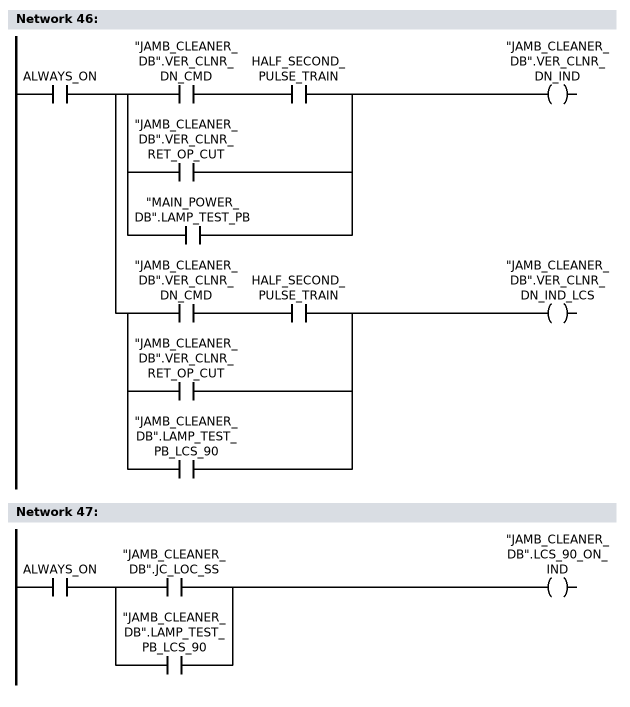
NETWORK
TITLE =
      A     "ALWAYS_ON";
      =     L 0.0;
      A     L 0.0;
      A(;
      A     "JAMB_CLEANER_DB".VER_CLNR_DN_CMD;
      A     "HALF_SECOND_PULSE_TRAIN";
      O     "JAMB_CLEANER_DB".VER_CLNR_RET_OP_CUT;
      O     "MAIN_POWER_DB".LAMP_TEST_PB;
      );
      =     "JAMB_CLEANER_DB".VER_CLNR_DN_IND;
      A     L 0.0;
      A(;
      A     "JAMB_CLEANER_DB".VER_CLNR_DN_CMD;
      A     "HALF_SECOND_PULSE_TRAIN";
      O     "JAMB_CLEANER_DB".VER_CLNR_RET_OP_CUT;
      O     "JAMB_CLEANER_DB".LAMP_TEST_PB_LCS_90;
      );
      =     "JAMB_CLEANER_DB".VER_CLNR_DN_IND_LCS;
NETWORK
TITLE =
      A     "ALWAYS_ON";
      A(;
      O     "JAMB_CLEANER_DB".JC_LOC_SS;
      O     "JAMB_CLEANER_DB".LAMP_TEST_PB_LCS_90;
      );
      =     "JAMB_CLEANER_DB".LCS_90_ON_IND;
END_FUNCTION

FUNCTION "COUNTER_THRUST_WEDGE" : VOID	// FC 17
AUTHOR : Kamillas
VERSION : 0.1
BEGIN
// (block stored without names or comments; labels and parameter names are numbered)
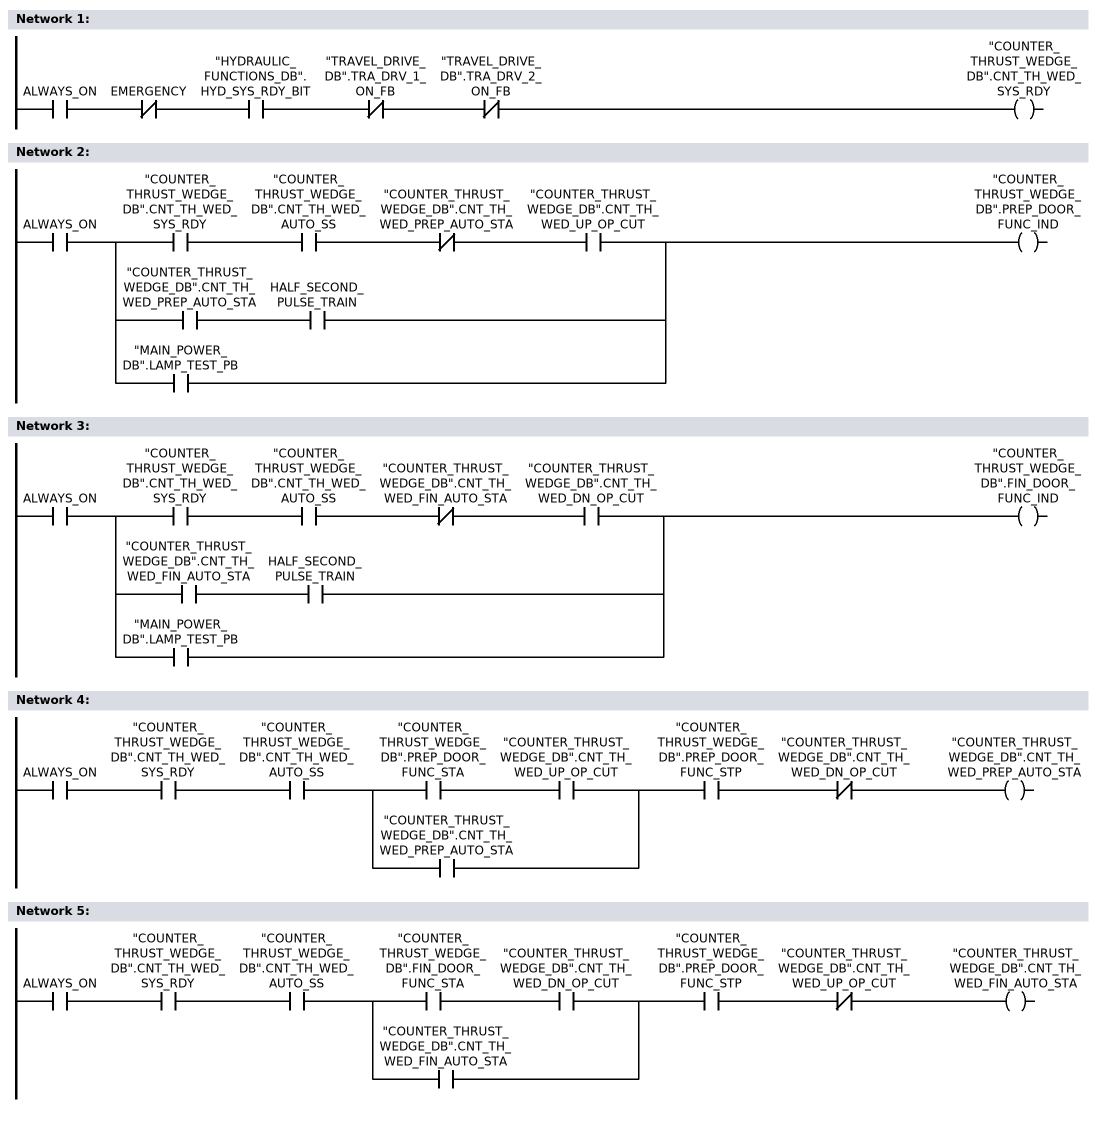
NETWORK
TITLE =
      A     "ALWAYS_ON";
      AN    "EMERGENCY";
      A     "HYDRAULIC_FUNCTIONS_DB".HYD_SYS_RDY_BIT;
      AN    "TRAVEL_DRIVE_DB".TRA_DRV_1_ON_FB;
      AN    "TRAVEL_DRIVE_DB".TRA_DRV_2_ON_FB;
      =     "COUNTER_THRUST_WEDGE_DB".CNT_TH_WED_SYS_RDY;
NETWORK
TITLE =
      A     "ALWAYS_ON";
      A(;
      A     "COUNTER_THRUST_WEDGE_DB".CNT_TH_WED_SYS_RDY;
      A     "COUNTER_THRUST_WEDGE_DB".CNT_TH_WED_AUTO_SS;
      AN    "COUNTER_THRUST_WEDGE_DB".CNT_TH_WED_PREP_AUTO_STA;
      A     "COUNTER_THRUST_WEDGE_DB".CNT_TH_WED_UP_OP_CUT;
      O;
      A     "COUNTER_THRUST_WEDGE_DB".CNT_TH_WED_PREP_AUTO_STA;
      A     "HALF_SECOND_PULSE_TRAIN";
      O     "MAIN_POWER_DB".LAMP_TEST_PB;
      );
      =     "COUNTER_THRUST_WEDGE_DB".PREP_DOOR_FUNC_IND;
NETWORK
TITLE =
      A     "ALWAYS_ON";
      A(;
      A     "COUNTER_THRUST_WEDGE_DB".CNT_TH_WED_SYS_RDY;
      A     "COUNTER_THRUST_WEDGE_DB".CNT_TH_WED_AUTO_SS;
      AN    "COUNTER_THRUST_WEDGE_DB".CNT_TH_WED_FIN_AUTO_STA;
      A     "COUNTER_THRUST_WEDGE_DB".CNT_TH_WED_DN_OP_CUT;
      O;
      A     "COUNTER_THRUST_WEDGE_DB".CNT_TH_WED_FIN_AUTO_STA;
      A     "HALF_SECOND_PULSE_TRAIN";
      O     "MAIN_POWER_DB".LAMP_TEST_PB;
      );
      =     "COUNTER_THRUST_WEDGE_DB".FIN_DOOR_FUNC_IND;
NETWORK
TITLE =
      A     "ALWAYS_ON";
      A     "COUNTER_THRUST_WEDGE_DB".CNT_TH_WED_SYS_RDY;
      A     "COUNTER_THRUST_WEDGE_DB".CNT_TH_WED_AUTO_SS;
      A(;
      A     "COUNTER_THRUST_WEDGE_DB".PREP_DOOR_FUNC_STA;
      A     "COUNTER_THRUST_WEDGE_DB".CNT_TH_WED_UP_OP_CUT;
      O     "COUNTER_THRUST_WEDGE_DB".CNT_TH_WED_PREP_AUTO_STA;
      );
      A     "COUNTER_THRUST_WEDGE_DB".PREP_DOOR_FUNC_STP;
      AN    "COUNTER_THRUST_WEDGE_DB".CNT_TH_WED_DN_OP_CUT;
      =     "COUNTER_THRUST_WEDGE_DB".CNT_TH_WED_PREP_AUTO_STA;
NETWORK
TITLE =
      A     "ALWAYS_ON";
      A     "COUNTER_THRUST_WEDGE_DB".CNT_TH_WED_SYS_RDY;
      A     "COUNTER_THRUST_WEDGE_DB".CNT_TH_WED_AUTO_SS;
      A(;
      A     "COUNTER_THRUST_WEDGE_DB".FIN_DOOR_FUNC_STA;
      A     "COUNTER_THRUST_WEDGE_DB".CNT_TH_WED_DN_OP_CUT;
      O     "COUNTER_THRUST_WEDGE_DB".CNT_TH_WED_FIN_AUTO_STA;
      );
      A     "COUNTER_THRUST_WEDGE_DB".PREP_DOOR_FUNC_STP;
      AN    "COUNTER_THRUST_WEDGE_DB".CNT_TH_WED_UP_OP_CUT;
      =     "COUNTER_THRUST_WEDGE_DB".CNT_TH_WED_FIN_AUTO_STA;
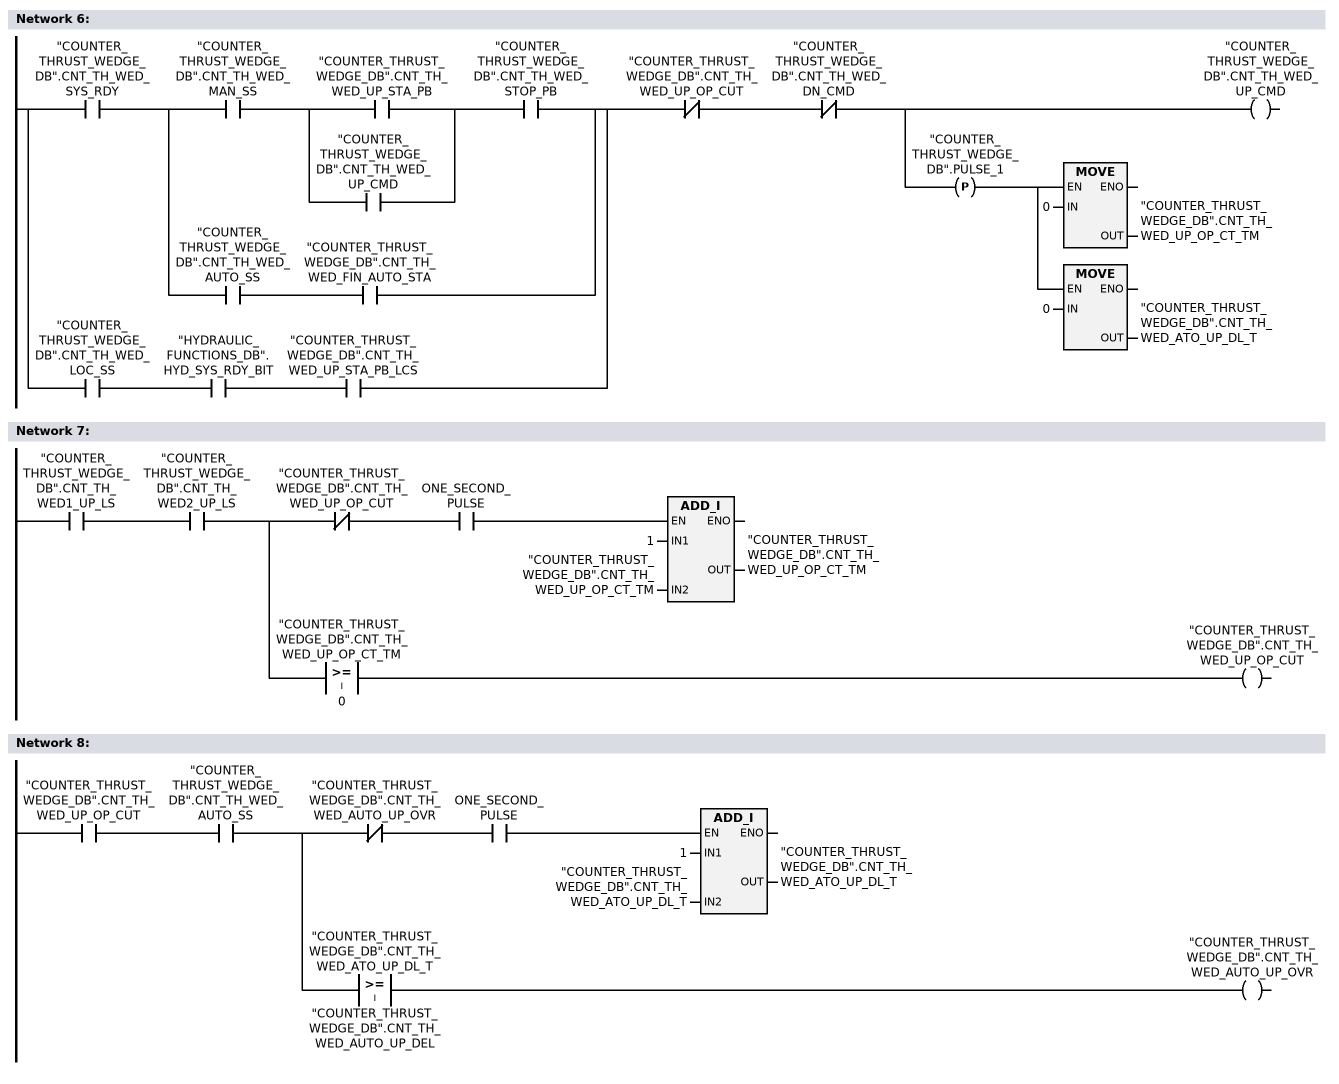
NETWORK
TITLE =
      A(;
      A     "COUNTER_THRUST_WEDGE_DB".CNT_TH_WED_SYS_RDY;
      A(;
      A     "COUNTER_THRUST_WEDGE_DB".CNT_TH_WED_MAN_SS;
      A(;
      O     "COUNTER_THRUST_WEDGE_DB".CNT_TH_WED_UP_STA_PB;
      O     "COUNTER_THRUST_WEDGE_DB".CNT_TH_WED_UP_CMD;
      );
      A     "COUNTER_THRUST_WEDGE_DB".CNT_TH_WED_STOP_PB;
      O;
      A     "COUNTER_THRUST_WEDGE_DB".CNT_TH_WED_AUTO_SS;
      A     "COUNTER_THRUST_WEDGE_DB".CNT_TH_WED_FIN_AUTO_STA;
      );
      O;
      A     "COUNTER_THRUST_WEDGE_DB".CNT_TH_WED_LOC_SS;
      A     "HYDRAULIC_FUNCTIONS_DB".HYD_SYS_RDY_BIT;
      A     "COUNTER_THRUST_WEDGE_DB".CNT_TH_WED_UP_STA_PB_LCS;
      );
      AN    "COUNTER_THRUST_WEDGE_DB".CNT_TH_WED_UP_OP_CUT;
      AN    "COUNTER_THRUST_WEDGE_DB".CNT_TH_WED_DN_CMD;
      =     L 0.0;
      A     L 0.0;
      BLD   102;
      =     "COUNTER_THRUST_WEDGE_DB".CNT_TH_WED_UP_CMD;
      A     L 0.0;
      FP    "COUNTER_THRUST_WEDGE_DB".PULSE_1;
      =     L 0.1;
      A     L 0.1;
      JNB   M001;
      L     0;
      T     "COUNTER_THRUST_WEDGE_DB".CNT_TH_WED_UP_OP_CT_TM;
M001: NOP   0;
      A     L 0.1;
      JNB   M002;
      L     0;
      T     "COUNTER_THRUST_WEDGE_DB".CNT_TH_WED_ATO_UP_DL_T;
M002: NOP   0;
NETWORK
TITLE =
      A     "COUNTER_THRUST_WEDGE_DB".CNT_TH_WED1_UP_LS;
      A     "COUNTER_THRUST_WEDGE_DB".CNT_TH_WED2_UP_LS;
      =     L 0.0;
      A     L 0.0;
      AN    "COUNTER_THRUST_WEDGE_DB".CNT_TH_WED_UP_OP_CUT;
      A     "ONE_SECOND_PULSE";
      JNB   M003;
      L     1;
      L     "COUNTER_THRUST_WEDGE_DB".CNT_TH_WED_UP_OP_CT_TM;
      +I;
      T     "COUNTER_THRUST_WEDGE_DB".CNT_TH_WED_UP_OP_CT_TM;
M003: NOP   0;
      A     L 0.0;
      A(;
      L     "COUNTER_THRUST_WEDGE_DB".CNT_TH_WED_UP_OP_CT_TM;
      L     0;
      >=I;
      );
      =     "COUNTER_THRUST_WEDGE_DB".CNT_TH_WED_UP_OP_CUT;
NETWORK
TITLE =
      A     "COUNTER_THRUST_WEDGE_DB".CNT_TH_WED_UP_OP_CUT;
      A     "COUNTER_THRUST_WEDGE_DB".CNT_TH_WED_AUTO_SS;
      =     L 0.0;
      A     L 0.0;
      AN    "COUNTER_THRUST_WEDGE_DB".CNT_TH_WED_AUTO_UP_OVR;
      A     "ONE_SECOND_PULSE";
      JNB   M004;
      L     1;
      L     "COUNTER_THRUST_WEDGE_DB".CNT_TH_WED_ATO_UP_DL_T;
      +I;
      T     "COUNTER_THRUST_WEDGE_DB".CNT_TH_WED_ATO_UP_DL_T;
M004: NOP   0;
      A     L 0.0;
      A(;
      L     "COUNTER_THRUST_WEDGE_DB".CNT_TH_WED_ATO_UP_DL_T;
      L     "COUNTER_THRUST_WEDGE_DB".CNT_TH_WED_AUTO_UP_DEL;
      >=I;
      );
      =     "COUNTER_THRUST_WEDGE_DB".CNT_TH_WED_AUTO_UP_OVR;
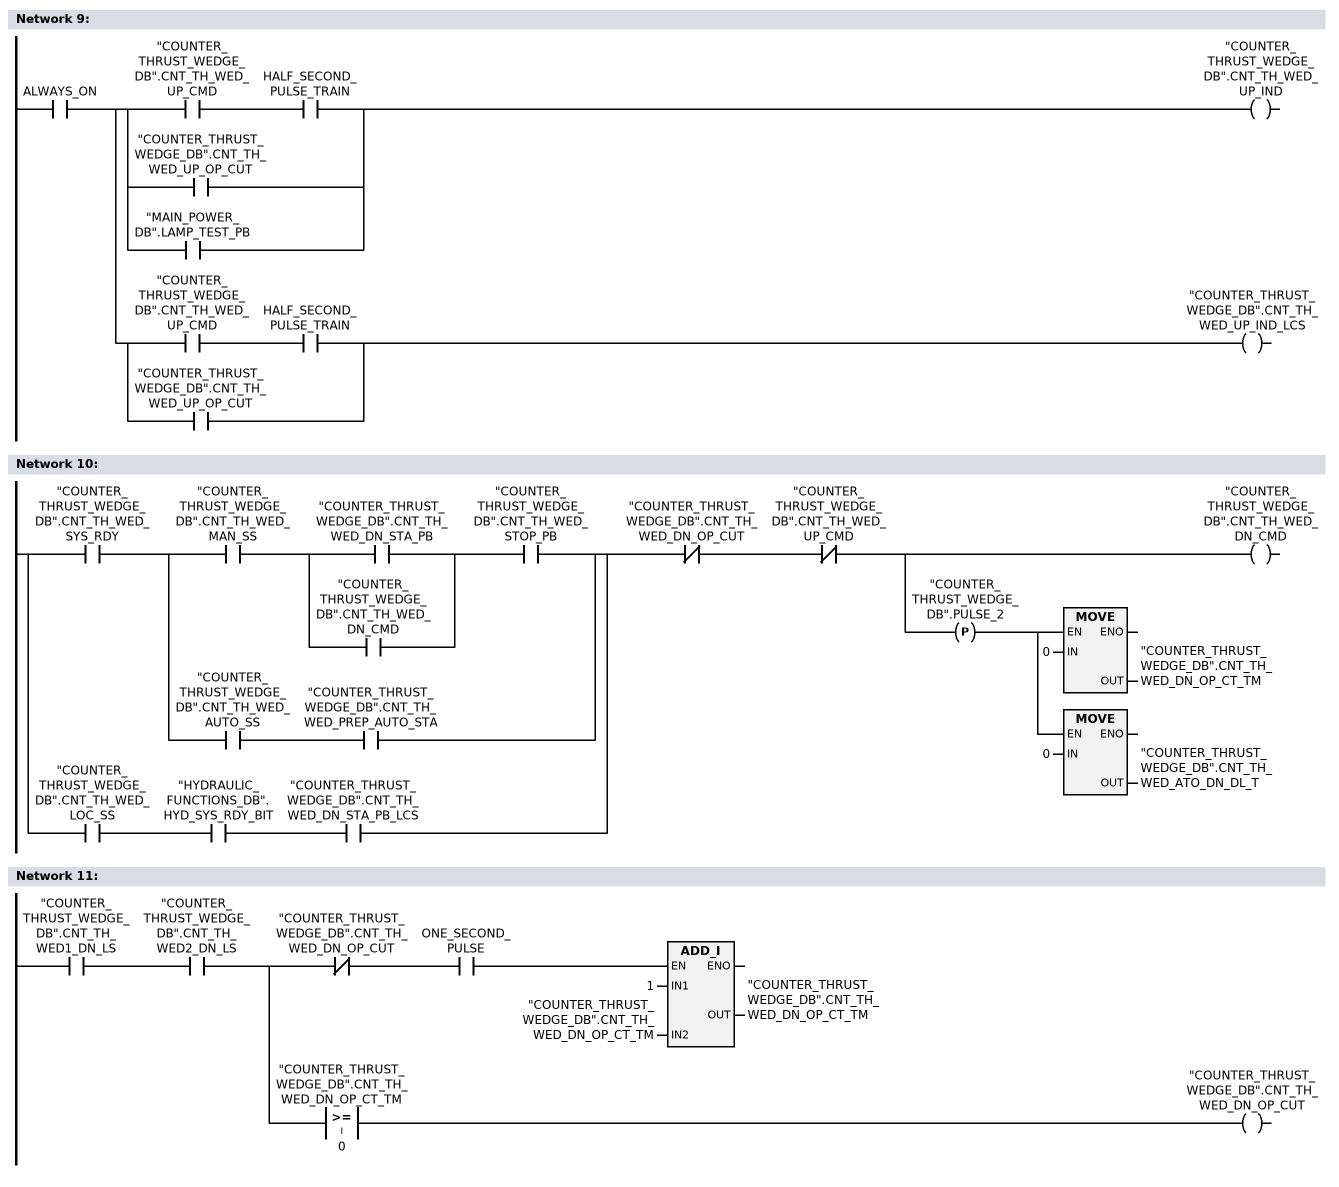
NETWORK
TITLE =
      A     "ALWAYS_ON";
      =     L 0.0;
      A     L 0.0;
      A(;
      A     "COUNTER_THRUST_WEDGE_DB".CNT_TH_WED_UP_CMD;
      A     "HALF_SECOND_PULSE_TRAIN";
      O     "COUNTER_THRUST_WEDGE_DB".CNT_TH_WED_UP_OP_CUT;
      O     "MAIN_POWER_DB".LAMP_TEST_PB;
      );
      =     "COUNTER_THRUST_WEDGE_DB".CNT_TH_WED_UP_IND;
      A     L 0.0;
      A(;
      A     "COUNTER_THRUST_WEDGE_DB".CNT_TH_WED_UP_CMD;
      A     "HALF_SECOND_PULSE_TRAIN";
      O     "COUNTER_THRUST_WEDGE_DB".CNT_TH_WED_UP_OP_CUT;
      );
      =     "COUNTER_THRUST_WEDGE_DB".CNT_TH_WED_UP_IND_LCS;
NETWORK
TITLE =
      A(;
      A     "COUNTER_THRUST_WEDGE_DB".CNT_TH_WED_SYS_RDY;
      A(;
      A     "COUNTER_THRUST_WEDGE_DB".CNT_TH_WED_MAN_SS;
      A(;
      O     "COUNTER_THRUST_WEDGE_DB".CNT_TH_WED_DN_STA_PB;
      O     "COUNTER_THRUST_WEDGE_DB".CNT_TH_WED_DN_CMD;
      );
      A     "COUNTER_THRUST_WEDGE_DB".CNT_TH_WED_STOP_PB;
      O;
      A     "COUNTER_THRUST_WEDGE_DB".CNT_TH_WED_AUTO_SS;
      A     "COUNTER_THRUST_WEDGE_DB".CNT_TH_WED_PREP_AUTO_STA;
      );
      O;
      A     "COUNTER_THRUST_WEDGE_DB".CNT_TH_WED_LOC_SS;
      A     "HYDRAULIC_FUNCTIONS_DB".HYD_SYS_RDY_BIT;
      A     "COUNTER_THRUST_WEDGE_DB".CNT_TH_WED_DN_STA_PB_LCS;
      );
      AN    "COUNTER_THRUST_WEDGE_DB".CNT_TH_WED_DN_OP_CUT;
      AN    "COUNTER_THRUST_WEDGE_DB".CNT_TH_WED_UP_CMD;
      =     L 0.0;
      A     L 0.0;
      BLD   102;
      =     "COUNTER_THRUST_WEDGE_DB".CNT_TH_WED_DN_CMD;
      A     L 0.0;
      FP    "COUNTER_THRUST_WEDGE_DB".PULSE_2;
      =     L 0.1;
      A     L 0.1;
      JNB   M005;
      L     0;
      T     "COUNTER_THRUST_WEDGE_DB".CNT_TH_WED_DN_OP_CT_TM;
M005: NOP   0;
      A     L 0.1;
      JNB   M006;
      L     0;
      T     "COUNTER_THRUST_WEDGE_DB".CNT_TH_WED_ATO_DN_DL_T;
M006: NOP   0;
NETWORK
TITLE =
      A     "COUNTER_THRUST_WEDGE_DB".CNT_TH_WED1_DN_LS;
      A     "COUNTER_THRUST_WEDGE_DB".CNT_TH_WED2_DN_LS;
      =     L 0.0;
      A     L 0.0;
      AN    "COUNTER_THRUST_WEDGE_DB".CNT_TH_WED_DN_OP_CUT;
      A     "ONE_SECOND_PULSE";
      JNB   M007;
      L     1;
      L     "COUNTER_THRUST_WEDGE_DB".CNT_TH_WED_DN_OP_CT_TM;
      +I;
      T     "COUNTER_THRUST_WEDGE_DB".CNT_TH_WED_DN_OP_CT_TM;
M007: NOP   0;
      A     L 0.0;
      A(;
      L     "COUNTER_THRUST_WEDGE_DB".CNT_TH_WED_DN_OP_CT_TM;
      L     0;
      >=I;
      );
      =     "COUNTER_THRUST_WEDGE_DB".CNT_TH_WED_DN_OP_CUT;
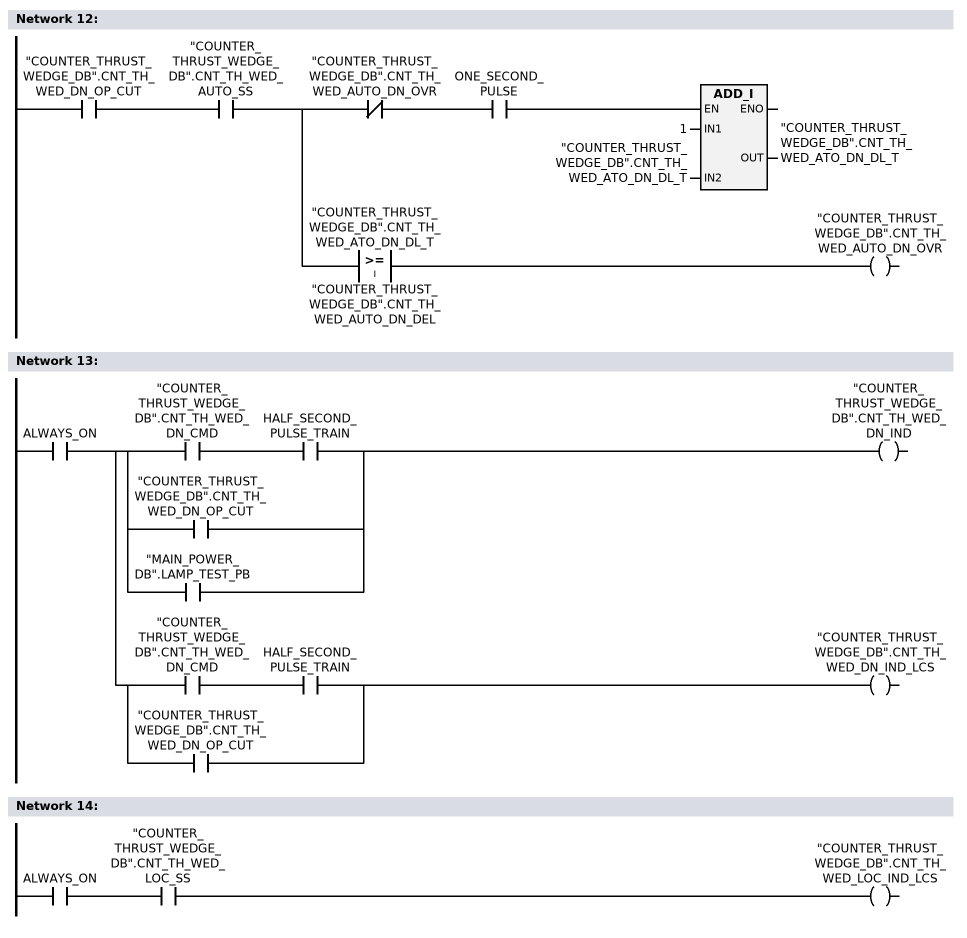
NETWORK
TITLE =
      A     "COUNTER_THRUST_WEDGE_DB".CNT_TH_WED_DN_OP_CUT;
      A     "COUNTER_THRUST_WEDGE_DB".CNT_TH_WED_AUTO_SS;
      =     L 0.0;
      A     L 0.0;
      AN    "COUNTER_THRUST_WEDGE_DB".CNT_TH_WED_AUTO_DN_OVR;
      A     "ONE_SECOND_PULSE";
      JNB   M008;
      L     1;
      L     "COUNTER_THRUST_WEDGE_DB".CNT_TH_WED_ATO_DN_DL_T;
      +I;
      T     "COUNTER_THRUST_WEDGE_DB".CNT_TH_WED_ATO_DN_DL_T;
M008: NOP   0;
      A     L 0.0;
      A(;
      L     "COUNTER_THRUST_WEDGE_DB".CNT_TH_WED_ATO_DN_DL_T;
      L     "COUNTER_THRUST_WEDGE_DB".CNT_TH_WED_AUTO_DN_DEL;
      >=I;
      );
      =     "COUNTER_THRUST_WEDGE_DB".CNT_TH_WED_AUTO_DN_OVR;
NETWORK
TITLE =
      A     "ALWAYS_ON";
      =     L 0.0;
      A     L 0.0;
      A(;
      A     "COUNTER_THRUST_WEDGE_DB".CNT_TH_WED_DN_CMD;
      A     "HALF_SECOND_PULSE_TRAIN";
      O     "COUNTER_THRUST_WEDGE_DB".CNT_TH_WED_DN_OP_CUT;
      O     "MAIN_POWER_DB".LAMP_TEST_PB;
      );
      =     "COUNTER_THRUST_WEDGE_DB".CNT_TH_WED_DN_IND;
      A     L 0.0;
      A(;
      A     "COUNTER_THRUST_WEDGE_DB".CNT_TH_WED_DN_CMD;
      A     "HALF_SECOND_PULSE_TRAIN";
      O     "COUNTER_THRUST_WEDGE_DB".CNT_TH_WED_DN_OP_CUT;
      );
      =     "COUNTER_THRUST_WEDGE_DB".CNT_TH_WED_DN_IND_LCS;
NETWORK
TITLE =
      A     "ALWAYS_ON";
      A     "COUNTER_THRUST_WEDGE_DB".CNT_TH_WED_LOC_SS;
      =     "COUNTER_THRUST_WEDGE_DB".CNT_TH_WED_LOC_IND_LCS;
END_FUNCTION

FUNCTION "COAL_SPILLAGE_SYSTEM" : VOID	// FC 18
AUTHOR : Kamillas
VERSION : 0.1
BEGIN
// (block stored without names or comments; labels and parameter names are numbered)
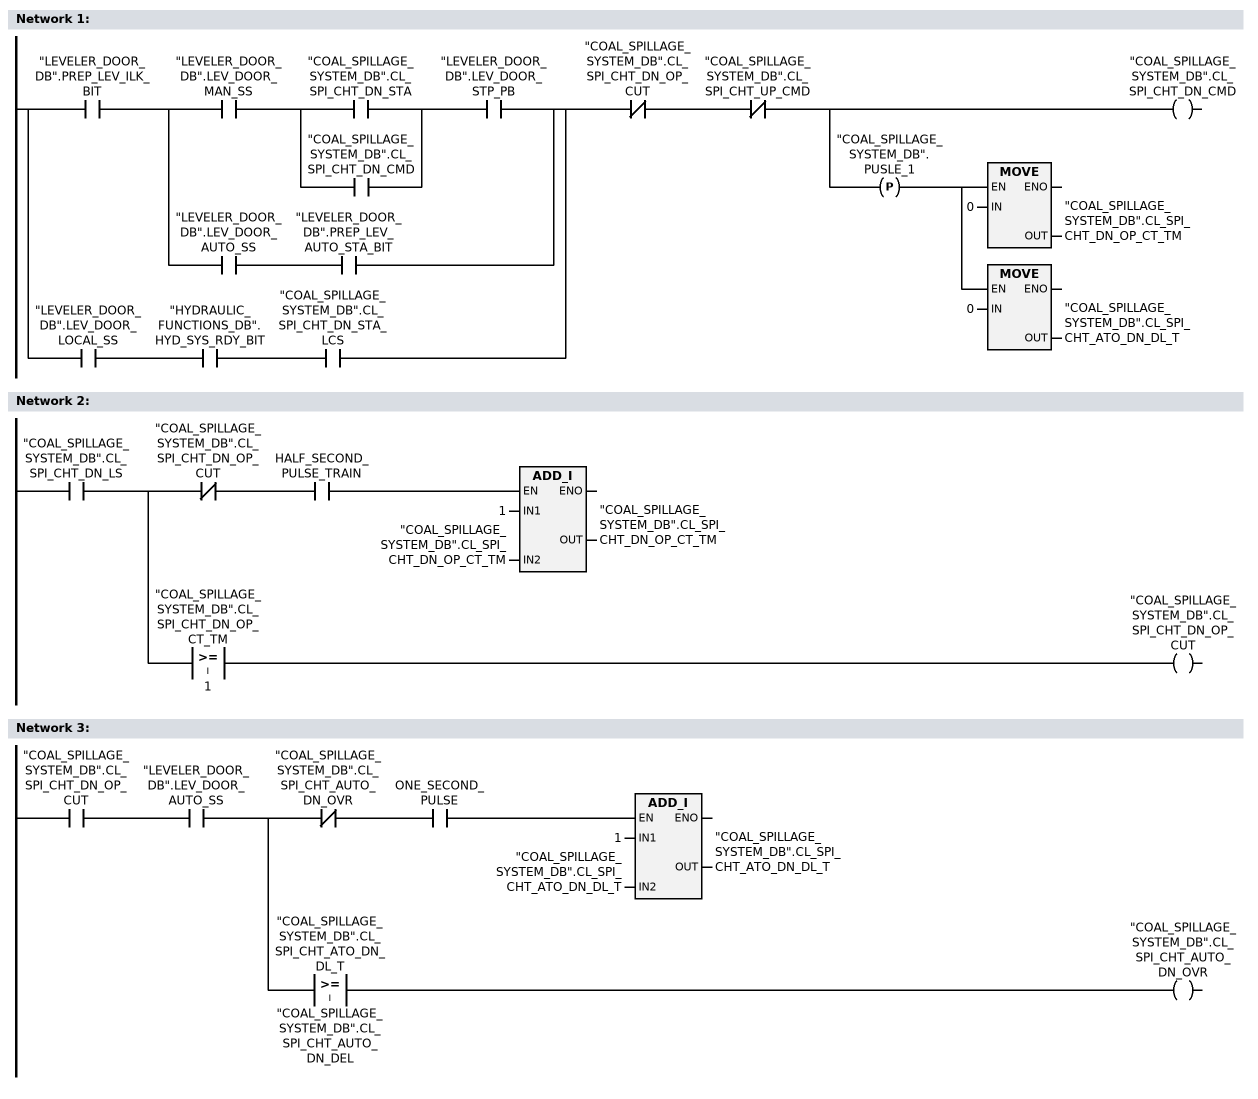
NETWORK
TITLE =
      A(;
      A     "LEVELER_DOOR_DB".PREP_LEV_ILK_BIT;
      A(;
      A     "LEVELER_DOOR_DB".LEV_DOOR_MAN_SS;
      A(;
      O     "COAL_SPILLAGE_SYSTEM_DB".CL_SPI_CHT_DN_STA;
      O     "COAL_SPILLAGE_SYSTEM_DB".CL_SPI_CHT_DN_CMD;
      );
      A     "LEVELER_DOOR_DB".LEV_DOOR_STP_PB;
      O;
      A     "LEVELER_DOOR_DB".LEV_DOOR_AUTO_SS;
      A     "LEVELER_DOOR_DB".PREP_LEV_AUTO_STA_BIT;
      );
      O;
      A     "LEVELER_DOOR_DB".LEV_DOOR_LOCAL_SS;
      A     "HYDRAULIC_FUNCTIONS_DB".HYD_SYS_RDY_BIT;
      A     "COAL_SPILLAGE_SYSTEM_DB".CL_SPI_CHT_DN_STA_LCS;
      );
      AN    "COAL_SPILLAGE_SYSTEM_DB".CL_SPI_CHT_DN_OP_CUT;
      AN    "COAL_SPILLAGE_SYSTEM_DB".CL_SPI_CHT_UP_CMD;
      =     L 0.0;
      A     L 0.0;
      BLD   102;
      =     "COAL_SPILLAGE_SYSTEM_DB".CL_SPI_CHT_DN_CMD;
      A     L 0.0;
      FP    "COAL_SPILLAGE_SYSTEM_DB".PUSLE_1;
      =     L 0.1;
      A     L 0.1;
      JNB   M001;
      L     0;
      T     "COAL_SPILLAGE_SYSTEM_DB".CL_SPI_CHT_DN_OP_CT_TM;
M001: NOP   0;
      A     L 0.1;
      JNB   M002;
      L     0;
      T     "COAL_SPILLAGE_SYSTEM_DB".CL_SPI_CHT_ATO_DN_DL_T;
M002: NOP   0;
NETWORK
TITLE =
      A     "COAL_SPILLAGE_SYSTEM_DB".CL_SPI_CHT_DN_LS;
      =     L 0.0;
      A     L 0.0;
      AN    "COAL_SPILLAGE_SYSTEM_DB".CL_SPI_CHT_DN_OP_CUT;
      A     "HALF_SECOND_PULSE_TRAIN";
      JNB   M003;
      L     1;
      L     "COAL_SPILLAGE_SYSTEM_DB".CL_SPI_CHT_DN_OP_CT_TM;
      +I;
      T     "COAL_SPILLAGE_SYSTEM_DB".CL_SPI_CHT_DN_OP_CT_TM;
M003: NOP   0;
      A     L 0.0;
      A(;
      L     "COAL_SPILLAGE_SYSTEM_DB".CL_SPI_CHT_DN_OP_CT_TM;
      L     1;
      >=I;
      );
      =     "COAL_SPILLAGE_SYSTEM_DB".CL_SPI_CHT_DN_OP_CUT;
NETWORK
TITLE =
      A     "COAL_SPILLAGE_SYSTEM_DB".CL_SPI_CHT_DN_OP_CUT;
      A     "LEVELER_DOOR_DB".LEV_DOOR_AUTO_SS;
      =     L 0.0;
      A     L 0.0;
      AN    "COAL_SPILLAGE_SYSTEM_DB".CL_SPI_CHT_AUTO_DN_OVR;
      A     "ONE_SECOND_PULSE";
      JNB   M004;
      L     1;
      L     "COAL_SPILLAGE_SYSTEM_DB".CL_SPI_CHT_ATO_DN_DL_T;
      +I;
      T     "COAL_SPILLAGE_SYSTEM_DB".CL_SPI_CHT_ATO_DN_DL_T;
M004: NOP   0;
      A     L 0.0;
      A(;
      L     "COAL_SPILLAGE_SYSTEM_DB".CL_SPI_CHT_ATO_DN_DL_T;
      L     "COAL_SPILLAGE_SYSTEM_DB".CL_SPI_CHT_AUTO_DN_DEL;
      >=I;
      );
      =     "COAL_SPILLAGE_SYSTEM_DB".CL_SPI_CHT_AUTO_DN_OVR;
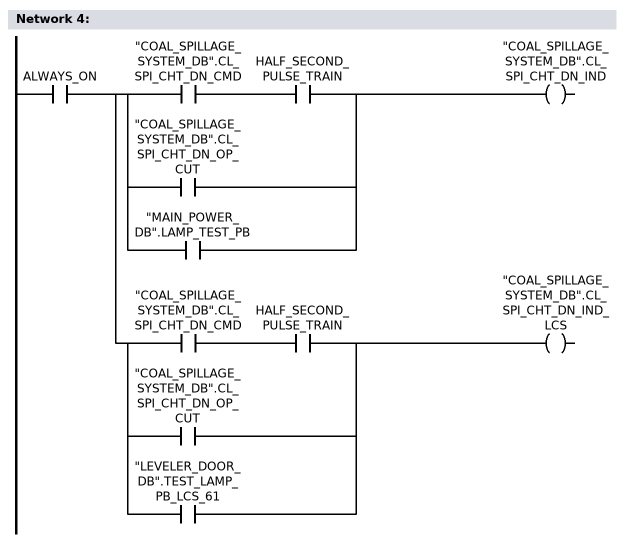
NETWORK
TITLE =
      A     "ALWAYS_ON";
      =     L 0.0;
      A     L 0.0;
      A(;
      A     "COAL_SPILLAGE_SYSTEM_DB".CL_SPI_CHT_DN_CMD;
      A     "HALF_SECOND_PULSE_TRAIN";
      O     "COAL_SPILLAGE_SYSTEM_DB".CL_SPI_CHT_DN_OP_CUT;
      O     "MAIN_POWER_DB".LAMP_TEST_PB;
      );
      =     "COAL_SPILLAGE_SYSTEM_DB".CL_SPI_CHT_DN_IND;
      A     L 0.0;
      A(;
      A     "COAL_SPILLAGE_SYSTEM_DB".CL_SPI_CHT_DN_CMD;
      A     "HALF_SECOND_PULSE_TRAIN";
      O     "COAL_SPILLAGE_SYSTEM_DB".CL_SPI_CHT_DN_OP_CUT;
      O     "LEVELER_DOOR_DB".TEST_LAMP_PB_LCS_61;
      );
      =     "COAL_SPILLAGE_SYSTEM_DB".CL_SPI_CHT_DN_IND_LCS;
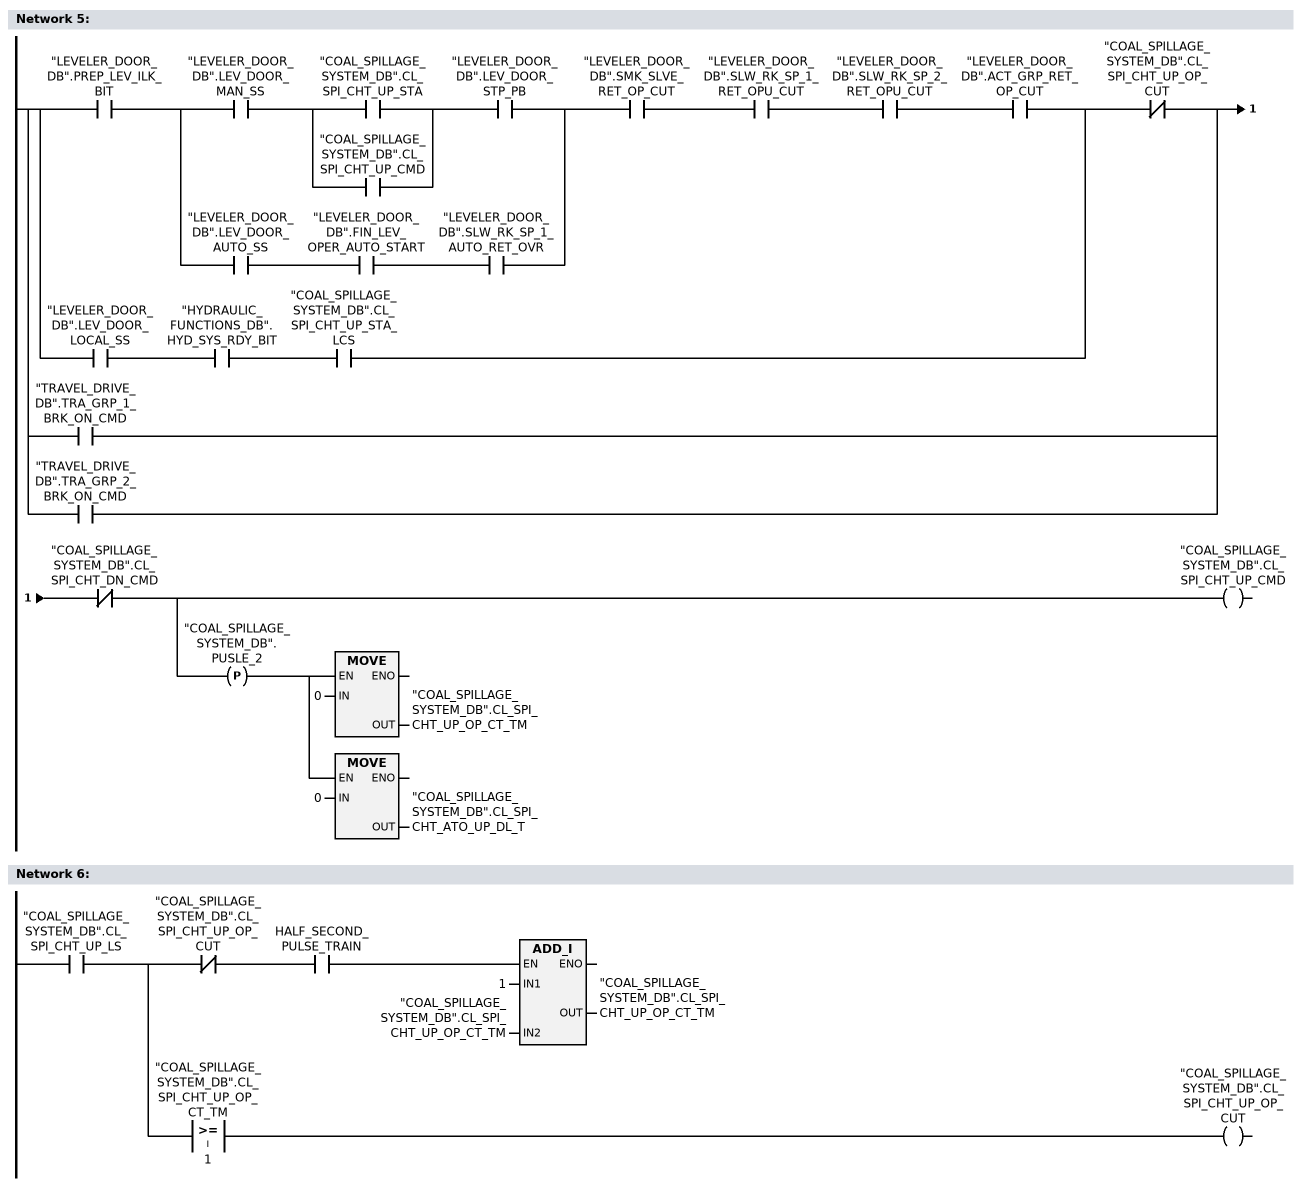
NETWORK
TITLE =
      A(;
      A(;
      A     "LEVELER_DOOR_DB".PREP_LEV_ILK_BIT;
      A(;
      A     "LEVELER_DOOR_DB".LEV_DOOR_MAN_SS;
      A(;
      O     "COAL_SPILLAGE_SYSTEM_DB".CL_SPI_CHT_UP_STA;
      O     "COAL_SPILLAGE_SYSTEM_DB".CL_SPI_CHT_UP_CMD;
      );
      A     "LEVELER_DOOR_DB".LEV_DOOR_STP_PB;
      O;
      A     "LEVELER_DOOR_DB".LEV_DOOR_AUTO_SS;
      A     "LEVELER_DOOR_DB".FIN_LEV_OPER_AUTO_START;
      A     "LEVELER_DOOR_DB".SLW_RK_SP_1_AUTO_RET_OVR;
      );
      A     "LEVELER_DOOR_DB".SMK_SLVE_RET_OP_CUT;
      A     "LEVELER_DOOR_DB".SLW_RK_SP_1_RET_OPU_CUT;
      A     "LEVELER_DOOR_DB".SLW_RK_SP_2_RET_OPU_CUT;
      A     "LEVELER_DOOR_DB".ACT_GRP_RET_OP_CUT;
      O;
      A     "LEVELER_DOOR_DB".LEV_DOOR_LOCAL_SS;
      A     "HYDRAULIC_FUNCTIONS_DB".HYD_SYS_RDY_BIT;
      A     "COAL_SPILLAGE_SYSTEM_DB".CL_SPI_CHT_UP_STA_LCS;
      );
      AN    "COAL_SPILLAGE_SYSTEM_DB".CL_SPI_CHT_UP_OP_CUT;
      O     "TRAVEL_DRIVE_DB".TRA_GRP_1_BRK_ON_CMD;
      O     "TRAVEL_DRIVE_DB".TRA_GRP_2_BRK_ON_CMD;
      );
      AN    "COAL_SPILLAGE_SYSTEM_DB".CL_SPI_CHT_DN_CMD;
      =     L 0.0;
      A     L 0.0;
      BLD   102;
      =     "COAL_SPILLAGE_SYSTEM_DB".CL_SPI_CHT_UP_CMD;
      A     L 0.0;
      FP    "COAL_SPILLAGE_SYSTEM_DB".PUSLE_2;
      =     L 0.1;
      A     L 0.1;
      JNB   M005;
      L     0;
      T     "COAL_SPILLAGE_SYSTEM_DB".CL_SPI_CHT_UP_OP_CT_TM;
M005: NOP   0;
      A     L 0.1;
      JNB   M006;
      L     0;
      T     "COAL_SPILLAGE_SYSTEM_DB".CL_SPI_CHT_ATO_UP_DL_T;
M006: NOP   0;
NETWORK
TITLE =
      A     "COAL_SPILLAGE_SYSTEM_DB".CL_SPI_CHT_UP_LS;
      =     L 0.0;
      A     L 0.0;
      AN    "COAL_SPILLAGE_SYSTEM_DB".CL_SPI_CHT_UP_OP_CUT;
      A     "HALF_SECOND_PULSE_TRAIN";
      JNB   M007;
      L     1;
      L     "COAL_SPILLAGE_SYSTEM_DB".CL_SPI_CHT_UP_OP_CT_TM;
      +I;
      T     "COAL_SPILLAGE_SYSTEM_DB".CL_SPI_CHT_UP_OP_CT_TM;
M007: NOP   0;
      A     L 0.0;
      A(;
      L     "COAL_SPILLAGE_SYSTEM_DB".CL_SPI_CHT_UP_OP_CT_TM;
      L     1;
      >=I;
      );
      =     "COAL_SPILLAGE_SYSTEM_DB".CL_SPI_CHT_UP_OP_CUT;
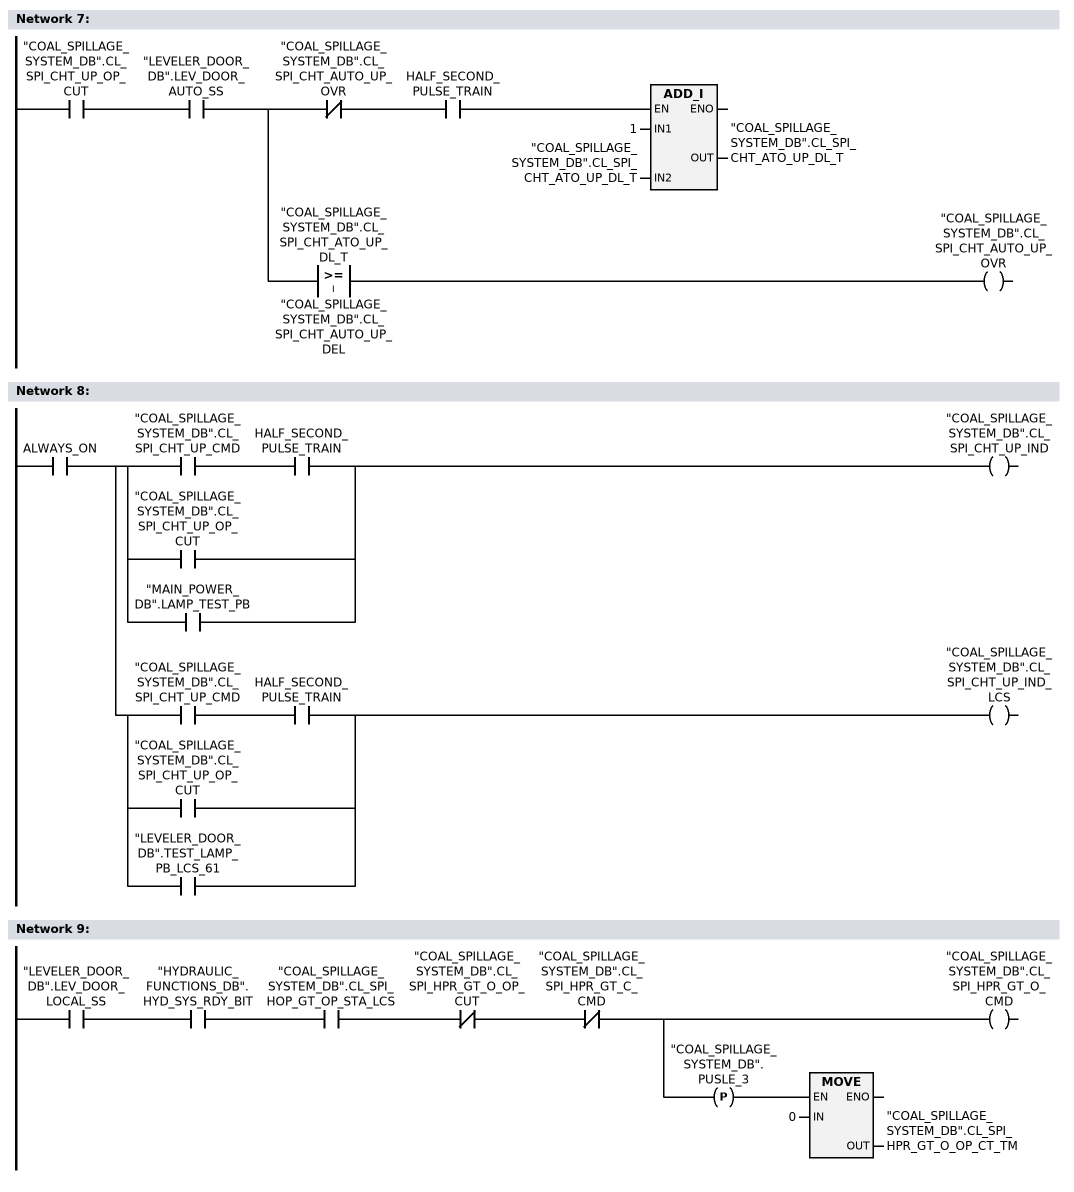
NETWORK
TITLE =
      A     "COAL_SPILLAGE_SYSTEM_DB".CL_SPI_CHT_UP_OP_CUT;
      A     "LEVELER_DOOR_DB".LEV_DOOR_AUTO_SS;
      =     L 0.0;
      A     L 0.0;
      AN    "COAL_SPILLAGE_SYSTEM_DB".CL_SPI_CHT_AUTO_UP_OVR;
      A     "HALF_SECOND_PULSE_TRAIN";
      JNB   M008;
      L     1;
      L     "COAL_SPILLAGE_SYSTEM_DB".CL_SPI_CHT_ATO_UP_DL_T;
      +I;
      T     "COAL_SPILLAGE_SYSTEM_DB".CL_SPI_CHT_ATO_UP_DL_T;
M008: NOP   0;
      A     L 0.0;
      A(;
      L     "COAL_SPILLAGE_SYSTEM_DB".CL_SPI_CHT_ATO_UP_DL_T;
      L     "COAL_SPILLAGE_SYSTEM_DB".CL_SPI_CHT_AUTO_UP_DEL;
      >=I;
      );
      =     "COAL_SPILLAGE_SYSTEM_DB".CL_SPI_CHT_AUTO_UP_OVR;
NETWORK
TITLE =
      A     "ALWAYS_ON";
      =     L 0.0;
      A     L 0.0;
      A(;
      A     "COAL_SPILLAGE_SYSTEM_DB".CL_SPI_CHT_UP_CMD;
      A     "HALF_SECOND_PULSE_TRAIN";
      O     "COAL_SPILLAGE_SYSTEM_DB".CL_SPI_CHT_UP_OP_CUT;
      O     "MAIN_POWER_DB".LAMP_TEST_PB;
      );
      =     "COAL_SPILLAGE_SYSTEM_DB".CL_SPI_CHT_UP_IND;
      A     L 0.0;
      A(;
      A     "COAL_SPILLAGE_SYSTEM_DB".CL_SPI_CHT_UP_CMD;
      A     "HALF_SECOND_PULSE_TRAIN";
      O     "COAL_SPILLAGE_SYSTEM_DB".CL_SPI_CHT_UP_OP_CUT;
      O     "LEVELER_DOOR_DB".TEST_LAMP_PB_LCS_61;
      );
      =     "COAL_SPILLAGE_SYSTEM_DB".CL_SPI_CHT_UP_IND_LCS;
NETWORK
TITLE =
      A     "LEVELER_DOOR_DB".LEV_DOOR_LOCAL_SS;
      A     "HYDRAULIC_FUNCTIONS_DB".HYD_SYS_RDY_BIT;
      A     "COAL_SPILLAGE_SYSTEM_DB".CL_SPI_HOP_GT_OP_STA_LCS;
      AN    "COAL_SPILLAGE_SYSTEM_DB".CL_SPI_HPR_GT_O_OP_CUT;
      AN    "COAL_SPILLAGE_SYSTEM_DB".CL_SPI_HPR_GT_C_CMD;
      =     L 0.0;
      A     L 0.0;
      BLD   102;
      =     "COAL_SPILLAGE_SYSTEM_DB".CL_SPI_HPR_GT_O_CMD;
      A     L 0.0;
      FP    "COAL_SPILLAGE_SYSTEM_DB".PUSLE_3;
      JNB   M009;
      L     0;
      T     "COAL_SPILLAGE_SYSTEM_DB".CL_SPI_HPR_GT_O_OP_CT_TM;
M009: NOP   0;
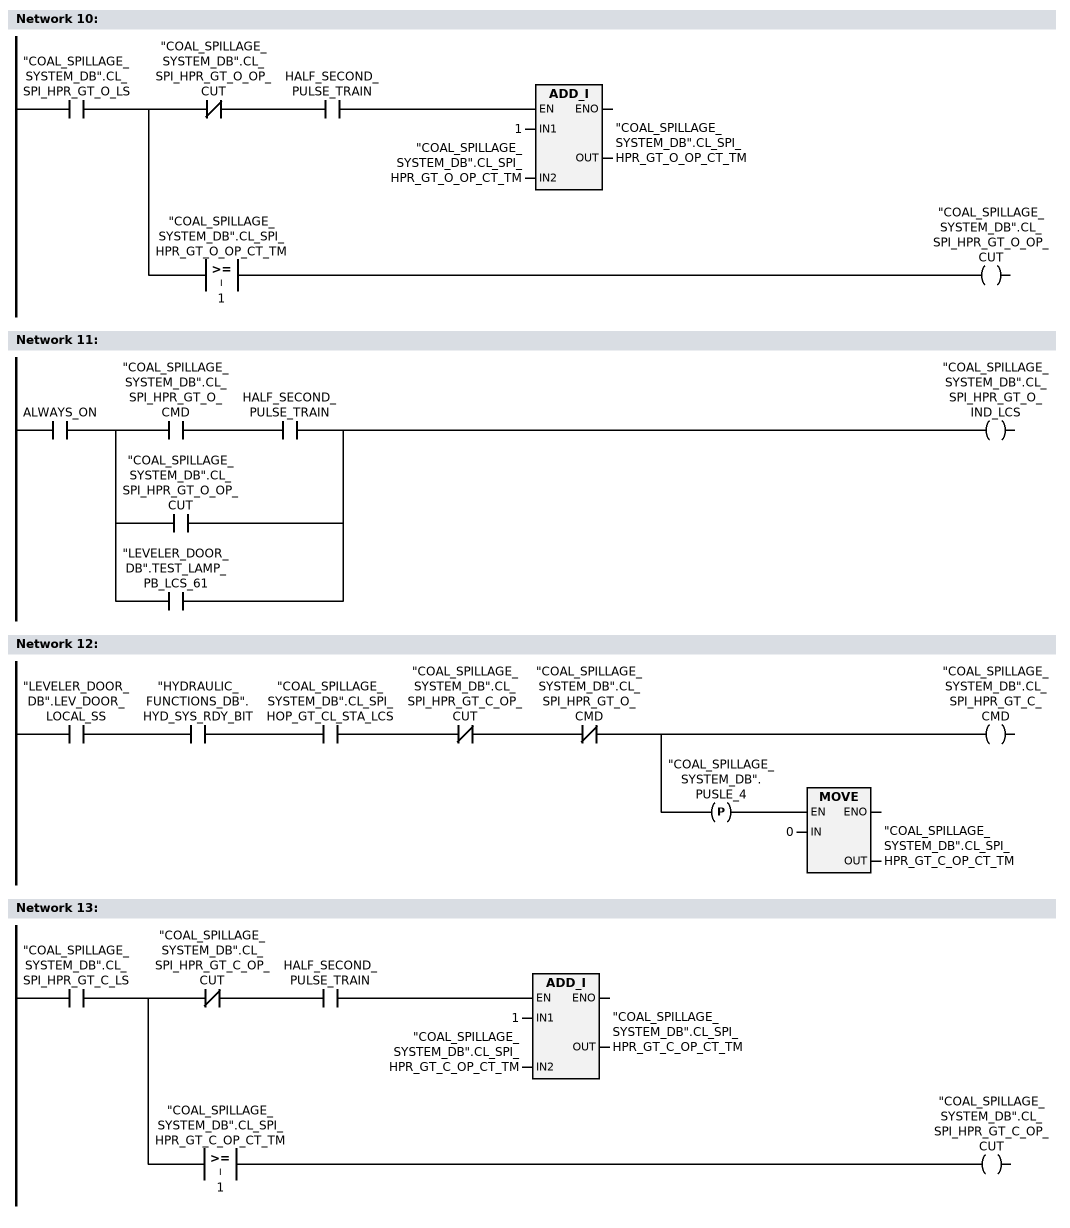
NETWORK
TITLE =
      A     "COAL_SPILLAGE_SYSTEM_DB".CL_SPI_HPR_GT_O_LS;
      =     L 0.0;
      A     L 0.0;
      AN    "COAL_SPILLAGE_SYSTEM_DB".CL_SPI_HPR_GT_O_OP_CUT;
      A     "HALF_SECOND_PULSE_TRAIN";
      JNB   M010;
      L     1;
      L     "COAL_SPILLAGE_SYSTEM_DB".CL_SPI_HPR_GT_O_OP_CT_TM;
      +I;
      T     "COAL_SPILLAGE_SYSTEM_DB".CL_SPI_HPR_GT_O_OP_CT_TM;
M010: NOP   0;
      A     L 0.0;
      A(;
      L     "COAL_SPILLAGE_SYSTEM_DB".CL_SPI_HPR_GT_O_OP_CT_TM;
      L     1;
      >=I;
      );
      =     "COAL_SPILLAGE_SYSTEM_DB".CL_SPI_HPR_GT_O_OP_CUT;
NETWORK
TITLE =
      A     "ALWAYS_ON";
      A(;
      A     "COAL_SPILLAGE_SYSTEM_DB".CL_SPI_HPR_GT_O_CMD;
      A     "HALF_SECOND_PULSE_TRAIN";
      O     "COAL_SPILLAGE_SYSTEM_DB".CL_SPI_HPR_GT_O_OP_CUT;
      O     "LEVELER_DOOR_DB".TEST_LAMP_PB_LCS_61;
      );
      =     "COAL_SPILLAGE_SYSTEM_DB".CL_SPI_HPR_GT_O_IND_LCS;
NETWORK
TITLE =
      A     "LEVELER_DOOR_DB".LEV_DOOR_LOCAL_SS;
      A     "HYDRAULIC_FUNCTIONS_DB".HYD_SYS_RDY_BIT;
      A     "COAL_SPILLAGE_SYSTEM_DB".CL_SPI_HOP_GT_CL_STA_LCS;
      AN    "COAL_SPILLAGE_SYSTEM_DB".CL_SPI_HPR_GT_C_OP_CUT;
      AN    "COAL_SPILLAGE_SYSTEM_DB".CL_SPI_HPR_GT_O_CMD;
      =     L 0.0;
      A     L 0.0;
      BLD   102;
      =     "COAL_SPILLAGE_SYSTEM_DB".CL_SPI_HPR_GT_C_CMD;
      A     L 0.0;
      FP    "COAL_SPILLAGE_SYSTEM_DB".PUSLE_4;
      JNB   M011;
      L     0;
      T     "COAL_SPILLAGE_SYSTEM_DB".CL_SPI_HPR_GT_C_OP_CT_TM;
M011: NOP   0;
NETWORK
TITLE =
      A     "COAL_SPILLAGE_SYSTEM_DB".CL_SPI_HPR_GT_C_LS;
      =     L 0.0;
      A     L 0.0;
      AN    "COAL_SPILLAGE_SYSTEM_DB".CL_SPI_HPR_GT_C_OP_CUT;
      A     "HALF_SECOND_PULSE_TRAIN";
      JNB   M012;
      L     1;
      L     "COAL_SPILLAGE_SYSTEM_DB".CL_SPI_HPR_GT_C_OP_CT_TM;
      +I;
      T     "COAL_SPILLAGE_SYSTEM_DB".CL_SPI_HPR_GT_C_OP_CT_TM;
M012: NOP   0;
      A     L 0.0;
      A(;
      L     "COAL_SPILLAGE_SYSTEM_DB".CL_SPI_HPR_GT_C_OP_CT_TM;
      L     1;
      >=I;
      );
      =     "COAL_SPILLAGE_SYSTEM_DB".CL_SPI_HPR_GT_C_OP_CUT;
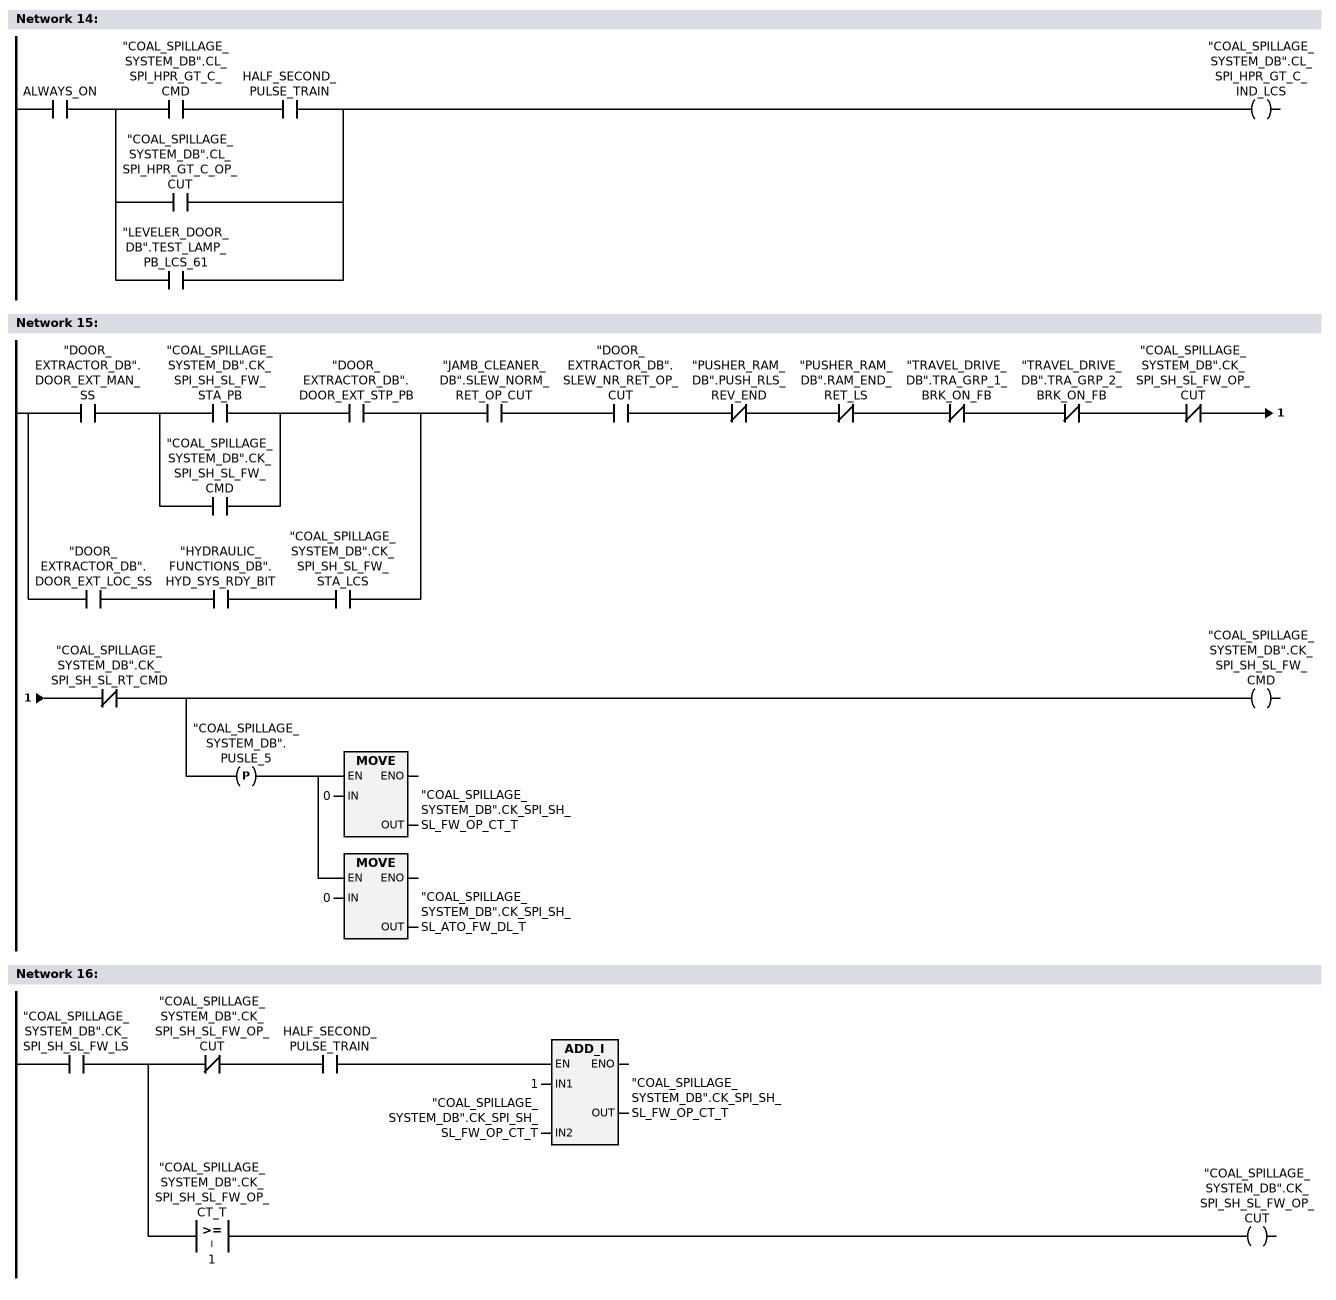
NETWORK
TITLE =
      A     "ALWAYS_ON";
      A(;
      A     "COAL_SPILLAGE_SYSTEM_DB".CL_SPI_HPR_GT_C_CMD;
      A     "HALF_SECOND_PULSE_TRAIN";
      O     "COAL_SPILLAGE_SYSTEM_DB".CL_SPI_HPR_GT_C_OP_CUT;
      O     "LEVELER_DOOR_DB".TEST_LAMP_PB_LCS_61;
      );
      =     "COAL_SPILLAGE_SYSTEM_DB".CL_SPI_HPR_GT_C_IND_LCS;
NETWORK
TITLE =
      A(;
      A     "DOOR_EXTRACTOR_DB".DOOR_EXT_MAN_SS;
      A(;
      O     "COAL_SPILLAGE_SYSTEM_DB".CK_SPI_SH_SL_FW_STA_PB;
      O     "COAL_SPILLAGE_SYSTEM_DB".CK_SPI_SH_SL_FW_CMD;
      );
      A     "DOOR_EXTRACTOR_DB".DOOR_EXT_STP_PB;
      O;
      A     "DOOR_EXTRACTOR_DB".DOOR_EXT_LOC_SS;
      A     "HYDRAULIC_FUNCTIONS_DB".HYD_SYS_RDY_BIT;
      A     "COAL_SPILLAGE_SYSTEM_DB".CK_SPI_SH_SL_FW_STA_LCS;
      );
      A     "JAMB_CLEANER_DB".SLEW_NORM_RET_OP_CUT;
      A     "DOOR_EXTRACTOR_DB".SLEW_NR_RET_OP_CUT;
      AN    "PUSHER_RAM_DB".PUSH_RLS_REV_END;
      AN    "PUSHER_RAM_DB".RAM_END_RET_LS;
      AN    "TRAVEL_DRIVE_DB".TRA_GRP_1_BRK_ON_FB;
      AN    "TRAVEL_DRIVE_DB".TRA_GRP_2_BRK_ON_FB;
      AN    "COAL_SPILLAGE_SYSTEM_DB".CK_SPI_SH_SL_FW_OP_CUT;
      AN    "COAL_SPILLAGE_SYSTEM_DB".CK_SPI_SH_SL_RT_CMD;
      =     L 0.0;
      A     L 0.0;
      BLD   102;
      =     "COAL_SPILLAGE_SYSTEM_DB".CK_SPI_SH_SL_FW_CMD;
      A     L 0.0;
      FP    "COAL_SPILLAGE_SYSTEM_DB".PUSLE_5;
      =     L 0.1;
      A     L 0.1;
      JNB   M013;
      L     0;
      T     "COAL_SPILLAGE_SYSTEM_DB".CK_SPI_SH_SL_FW_OP_CT_T;
M013: NOP   0;
      A     L 0.1;
      JNB   M014;
      L     0;
      T     "COAL_SPILLAGE_SYSTEM_DB".CK_SPI_SH_SL_ATO_FW_DL_T;
M014: NOP   0;
NETWORK
TITLE =
      A     "COAL_SPILLAGE_SYSTEM_DB".CK_SPI_SH_SL_FW_LS;
      =     L 0.0;
      A     L 0.0;
      AN    "COAL_SPILLAGE_SYSTEM_DB".CK_SPI_SH_SL_FW_OP_CUT;
      A     "HALF_SECOND_PULSE_TRAIN";
      JNB   M015;
      L     1;
      L     "COAL_SPILLAGE_SYSTEM_DB".CK_SPI_SH_SL_FW_OP_CT_T;
      +I;
      T     "COAL_SPILLAGE_SYSTEM_DB".CK_SPI_SH_SL_FW_OP_CT_T;
M015: NOP   0;
      A     L 0.0;
      A(;
      L     "COAL_SPILLAGE_SYSTEM_DB".CK_SPI_SH_SL_FW_OP_CT_T;
      L     1;
      >=I;
      );
      =     "COAL_SPILLAGE_SYSTEM_DB".CK_SPI_SH_SL_FW_OP_CUT;
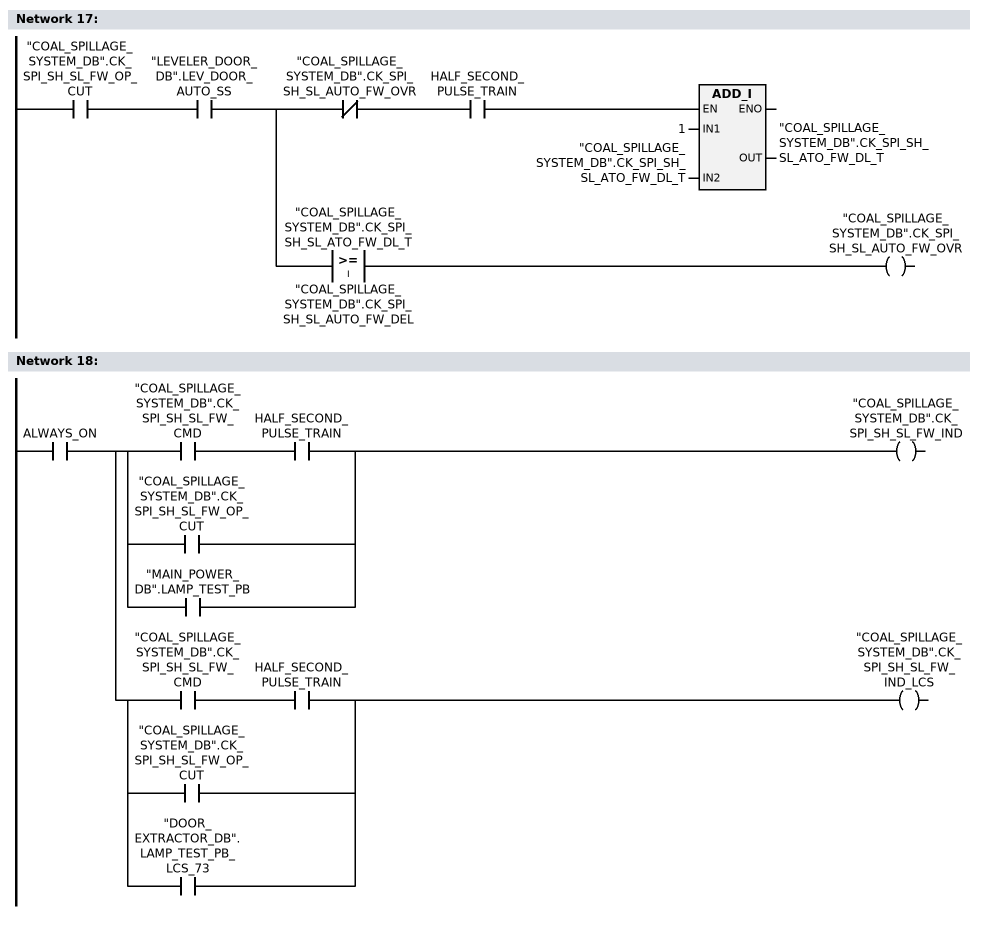
NETWORK
TITLE =
      A     "COAL_SPILLAGE_SYSTEM_DB".CK_SPI_SH_SL_FW_OP_CUT;
      A     "LEVELER_DOOR_DB".LEV_DOOR_AUTO_SS;
      =     L 0.0;
      A     L 0.0;
      AN    "COAL_SPILLAGE_SYSTEM_DB".CK_SPI_SH_SL_AUTO_FW_OVR;
      A     "HALF_SECOND_PULSE_TRAIN";
      JNB   M016;
      L     1;
      L     "COAL_SPILLAGE_SYSTEM_DB".CK_SPI_SH_SL_ATO_FW_DL_T;
      +I;
      T     "COAL_SPILLAGE_SYSTEM_DB".CK_SPI_SH_SL_ATO_FW_DL_T;
M016: NOP   0;
      A     L 0.0;
      A(;
      L     "COAL_SPILLAGE_SYSTEM_DB".CK_SPI_SH_SL_ATO_FW_DL_T;
      L     "COAL_SPILLAGE_SYSTEM_DB".CK_SPI_SH_SL_AUTO_FW_DEL;
      >=I;
      );
      =     "COAL_SPILLAGE_SYSTEM_DB".CK_SPI_SH_SL_AUTO_FW_OVR;
NETWORK
TITLE =
      A     "ALWAYS_ON";
      =     L 0.0;
      A     L 0.0;
      A(;
      A     "COAL_SPILLAGE_SYSTEM_DB".CK_SPI_SH_SL_FW_CMD;
      A     "HALF_SECOND_PULSE_TRAIN";
      O     "COAL_SPILLAGE_SYSTEM_DB".CK_SPI_SH_SL_FW_OP_CUT;
      O     "MAIN_POWER_DB".LAMP_TEST_PB;
      );
      =     "COAL_SPILLAGE_SYSTEM_DB".CK_SPI_SH_SL_FW_IND;
      A     L 0.0;
      A(;
      A     "COAL_SPILLAGE_SYSTEM_DB".CK_SPI_SH_SL_FW_CMD;
      A     "HALF_SECOND_PULSE_TRAIN";
      O     "COAL_SPILLAGE_SYSTEM_DB".CK_SPI_SH_SL_FW_OP_CUT;
      O     "DOOR_EXTRACTOR_DB".LAMP_TEST_PB_LCS_73;
      );
      =     "COAL_SPILLAGE_SYSTEM_DB".CK_SPI_SH_SL_FW_IND_LCS;
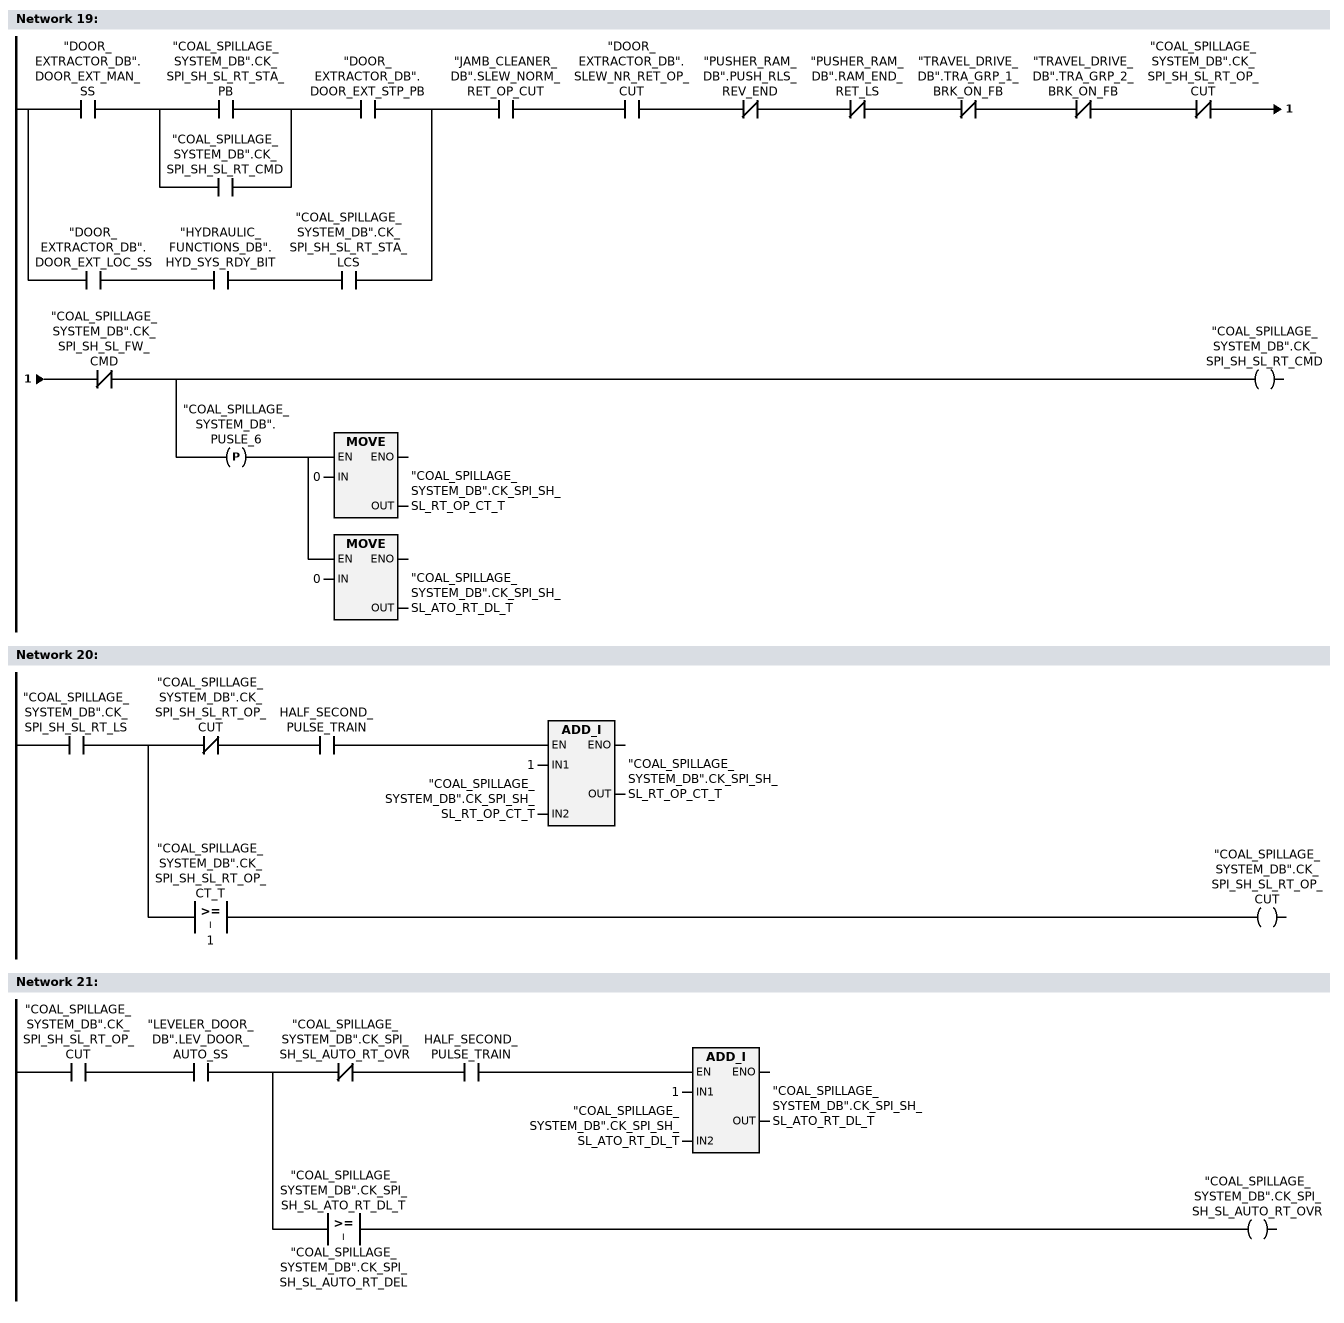
NETWORK
TITLE =
      A(;
      A     "DOOR_EXTRACTOR_DB".DOOR_EXT_MAN_SS;
      A(;
      O     "COAL_SPILLAGE_SYSTEM_DB".CK_SPI_SH_SL_RT_STA_PB;
      O     "COAL_SPILLAGE_SYSTEM_DB".CK_SPI_SH_SL_RT_CMD;
      );
      A     "DOOR_EXTRACTOR_DB".DOOR_EXT_STP_PB;
      O;
      A     "DOOR_EXTRACTOR_DB".DOOR_EXT_LOC_SS;
      A     "HYDRAULIC_FUNCTIONS_DB".HYD_SYS_RDY_BIT;
      A     "COAL_SPILLAGE_SYSTEM_DB".CK_SPI_SH_SL_RT_STA_LCS;
      );
      A     "JAMB_CLEANER_DB".SLEW_NORM_RET_OP_CUT;
      A     "DOOR_EXTRACTOR_DB".SLEW_NR_RET_OP_CUT;
      AN    "PUSHER_RAM_DB".PUSH_RLS_REV_END;
      AN    "PUSHER_RAM_DB".RAM_END_RET_LS;
      AN    "TRAVEL_DRIVE_DB".TRA_GRP_1_BRK_ON_FB;
      AN    "TRAVEL_DRIVE_DB".TRA_GRP_2_BRK_ON_FB;
      AN    "COAL_SPILLAGE_SYSTEM_DB".CK_SPI_SH_SL_RT_OP_CUT;
      AN    "COAL_SPILLAGE_SYSTEM_DB".CK_SPI_SH_SL_FW_CMD;
      =     L 0.0;
      A     L 0.0;
      BLD   102;
      =     "COAL_SPILLAGE_SYSTEM_DB".CK_SPI_SH_SL_RT_CMD;
      A     L 0.0;
      FP    "COAL_SPILLAGE_SYSTEM_DB".PUSLE_6;
      =     L 0.1;
      A     L 0.1;
      JNB   M017;
      L     0;
      T     "COAL_SPILLAGE_SYSTEM_DB".CK_SPI_SH_SL_RT_OP_CT_T;
M017: NOP   0;
      A     L 0.1;
      JNB   M018;
      L     0;
      T     "COAL_SPILLAGE_SYSTEM_DB".CK_SPI_SH_SL_ATO_RT_DL_T;
M018: NOP   0;
NETWORK
TITLE =
      A     "COAL_SPILLAGE_SYSTEM_DB".CK_SPI_SH_SL_RT_LS;
      =     L 0.0;
      A     L 0.0;
      AN    "COAL_SPILLAGE_SYSTEM_DB".CK_SPI_SH_SL_RT_OP_CUT;
      A     "HALF_SECOND_PULSE_TRAIN";
      JNB   M019;
      L     1;
      L     "COAL_SPILLAGE_SYSTEM_DB".CK_SPI_SH_SL_RT_OP_CT_T;
      +I;
      T     "COAL_SPILLAGE_SYSTEM_DB".CK_SPI_SH_SL_RT_OP_CT_T;
M019: NOP   0;
      A     L 0.0;
      A(;
      L     "COAL_SPILLAGE_SYSTEM_DB".CK_SPI_SH_SL_RT_OP_CT_T;
      L     1;
      >=I;
      );
      =     "COAL_SPILLAGE_SYSTEM_DB".CK_SPI_SH_SL_RT_OP_CUT;
NETWORK
TITLE =
      A     "COAL_SPILLAGE_SYSTEM_DB".CK_SPI_SH_SL_RT_OP_CUT;
      A     "LEVELER_DOOR_DB".LEV_DOOR_AUTO_SS;
      =     L 0.0;
      A     L 0.0;
      AN    "COAL_SPILLAGE_SYSTEM_DB".CK_SPI_SH_SL_AUTO_RT_OVR;
      A     "HALF_SECOND_PULSE_TRAIN";
      JNB   M020;
      L     1;
      L     "COAL_SPILLAGE_SYSTEM_DB".CK_SPI_SH_SL_ATO_RT_DL_T;
      +I;
      T     "COAL_SPILLAGE_SYSTEM_DB".CK_SPI_SH_SL_ATO_RT_DL_T;
M020: NOP   0;
      A     L 0.0;
      A(;
      L     "COAL_SPILLAGE_SYSTEM_DB".CK_SPI_SH_SL_ATO_RT_DL_T;
      L     "COAL_SPILLAGE_SYSTEM_DB".CK_SPI_SH_SL_AUTO_RT_DEL;
      >=I;
      );
      =     "COAL_SPILLAGE_SYSTEM_DB".CK_SPI_SH_SL_AUTO_RT_OVR;
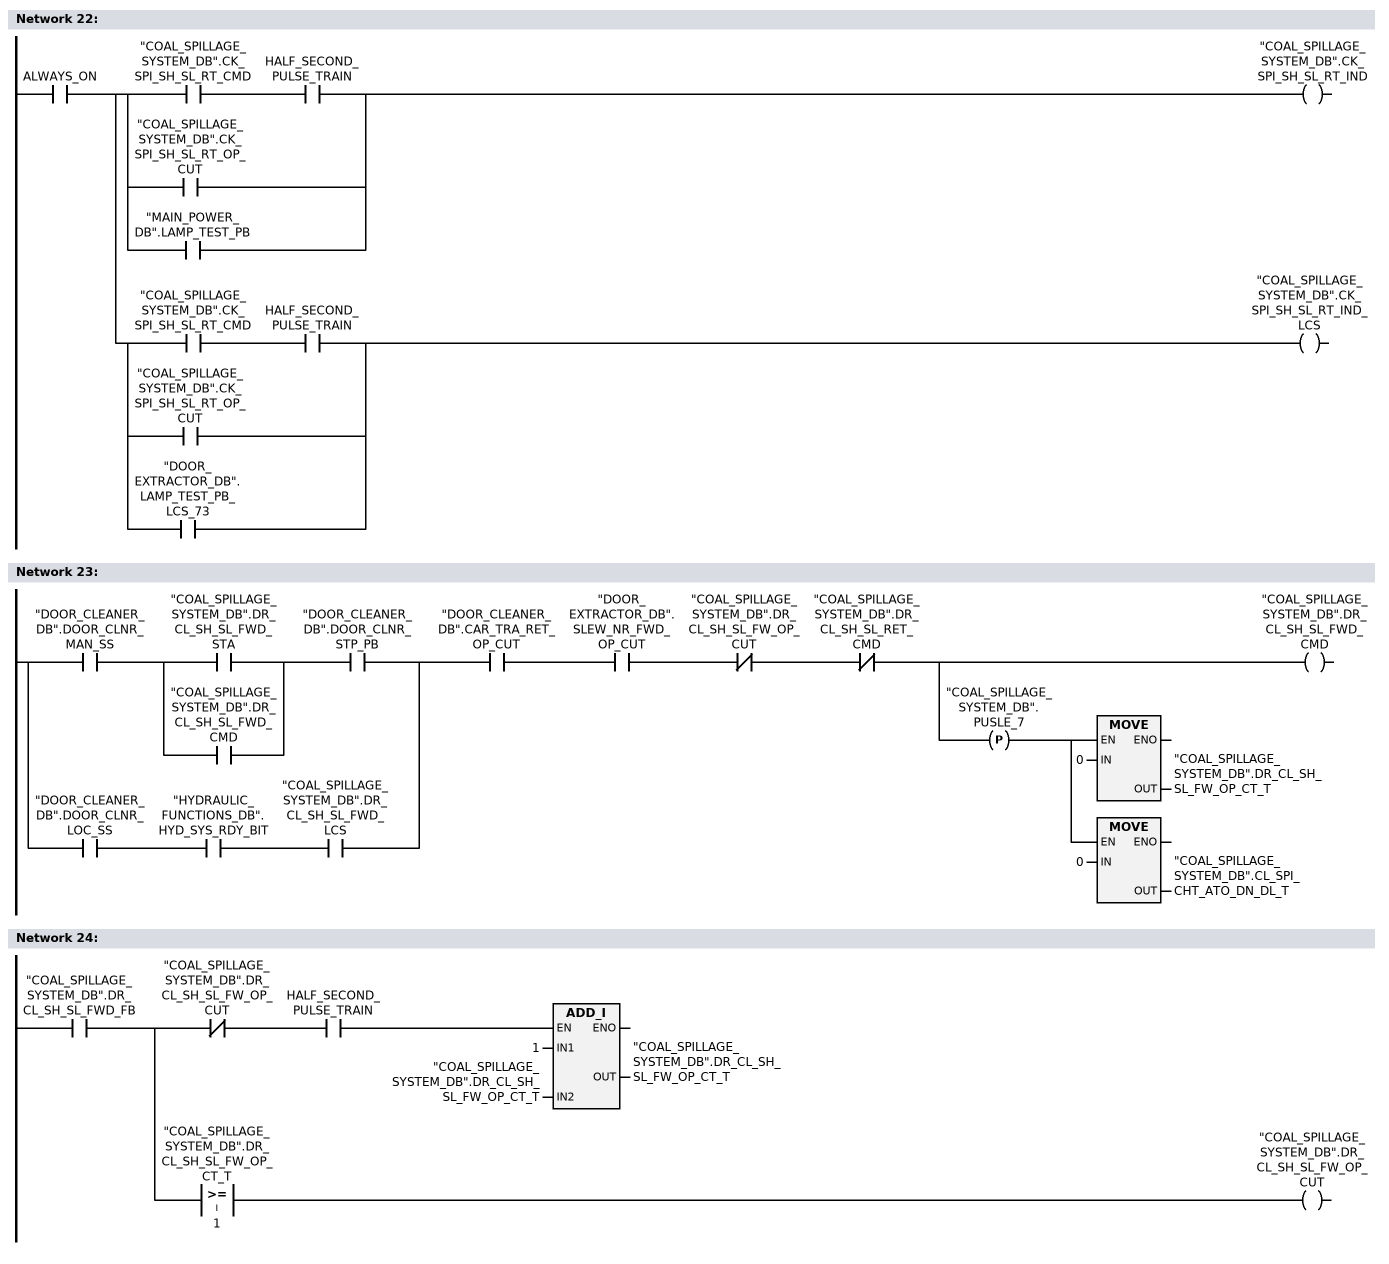
NETWORK
TITLE =
      A     "ALWAYS_ON";
      =     L 0.0;
      A     L 0.0;
      A(;
      A     "COAL_SPILLAGE_SYSTEM_DB".CK_SPI_SH_SL_RT_CMD;
      A     "HALF_SECOND_PULSE_TRAIN";
      O     "COAL_SPILLAGE_SYSTEM_DB".CK_SPI_SH_SL_RT_OP_CUT;
      O     "MAIN_POWER_DB".LAMP_TEST_PB;
      );
      =     "COAL_SPILLAGE_SYSTEM_DB".CK_SPI_SH_SL_RT_IND;
      A     L 0.0;
      A(;
      A     "COAL_SPILLAGE_SYSTEM_DB".CK_SPI_SH_SL_RT_CMD;
      A     "HALF_SECOND_PULSE_TRAIN";
      O     "COAL_SPILLAGE_SYSTEM_DB".CK_SPI_SH_SL_RT_OP_CUT;
      O     "DOOR_EXTRACTOR_DB".LAMP_TEST_PB_LCS_73;
      );
      =     "COAL_SPILLAGE_SYSTEM_DB".CK_SPI_SH_SL_RT_IND_LCS;
NETWORK
TITLE =
      A(;
      A     "DOOR_CLEANER_DB".DOOR_CLNR_MAN_SS;
      A(;
      O     "COAL_SPILLAGE_SYSTEM_DB".DR_CL_SH_SL_FWD_STA;
      O     "COAL_SPILLAGE_SYSTEM_DB".DR_CL_SH_SL_FWD_CMD;
      );
      A     "DOOR_CLEANER_DB".DOOR_CLNR_STP_PB;
      O;
      A     "DOOR_CLEANER_DB".DOOR_CLNR_LOC_SS;
      A     "HYDRAULIC_FUNCTIONS_DB".HYD_SYS_RDY_BIT;
      A     "COAL_SPILLAGE_SYSTEM_DB".DR_CL_SH_SL_FWD_LCS;
      );
      A     "DOOR_CLEANER_DB".CAR_TRA_RET_OP_CUT;
      A     "DOOR_EXTRACTOR_DB".SLEW_NR_FWD_OP_CUT;
      AN    "COAL_SPILLAGE_SYSTEM_DB".DR_CL_SH_SL_FW_OP_CUT;
      AN    "COAL_SPILLAGE_SYSTEM_DB".DR_CL_SH_SL_RET_CMD;
      =     L 0.0;
      A     L 0.0;
      BLD   102;
      =     "COAL_SPILLAGE_SYSTEM_DB".DR_CL_SH_SL_FWD_CMD;
      A     L 0.0;
      FP    "COAL_SPILLAGE_SYSTEM_DB".PUSLE_7;
      =     L 0.1;
      A     L 0.1;
      JNB   M021;
      L     0;
      T     "COAL_SPILLAGE_SYSTEM_DB".DR_CL_SH_SL_FW_OP_CT_T;
M021: NOP   0;
      A     L 0.1;
      JNB   M022;
      L     0;
      T     "COAL_SPILLAGE_SYSTEM_DB".CL_SPI_CHT_ATO_DN_DL_T;
M022: NOP   0;
NETWORK
TITLE =
      A     "COAL_SPILLAGE_SYSTEM_DB".DR_CL_SH_SL_FWD_FB;
      =     L 0.0;
      A     L 0.0;
      AN    "COAL_SPILLAGE_SYSTEM_DB".DR_CL_SH_SL_FW_OP_CUT;
      A     "HALF_SECOND_PULSE_TRAIN";
      JNB   M023;
      L     1;
      L     "COAL_SPILLAGE_SYSTEM_DB".DR_CL_SH_SL_FW_OP_CT_T;
      +I;
      T     "COAL_SPILLAGE_SYSTEM_DB".DR_CL_SH_SL_FW_OP_CT_T;
M023: NOP   0;
      A     L 0.0;
      A(;
      L     "COAL_SPILLAGE_SYSTEM_DB".DR_CL_SH_SL_FW_OP_CT_T;
      L     1;
      >=I;
      );
      =     "COAL_SPILLAGE_SYSTEM_DB".DR_CL_SH_SL_FW_OP_CUT;
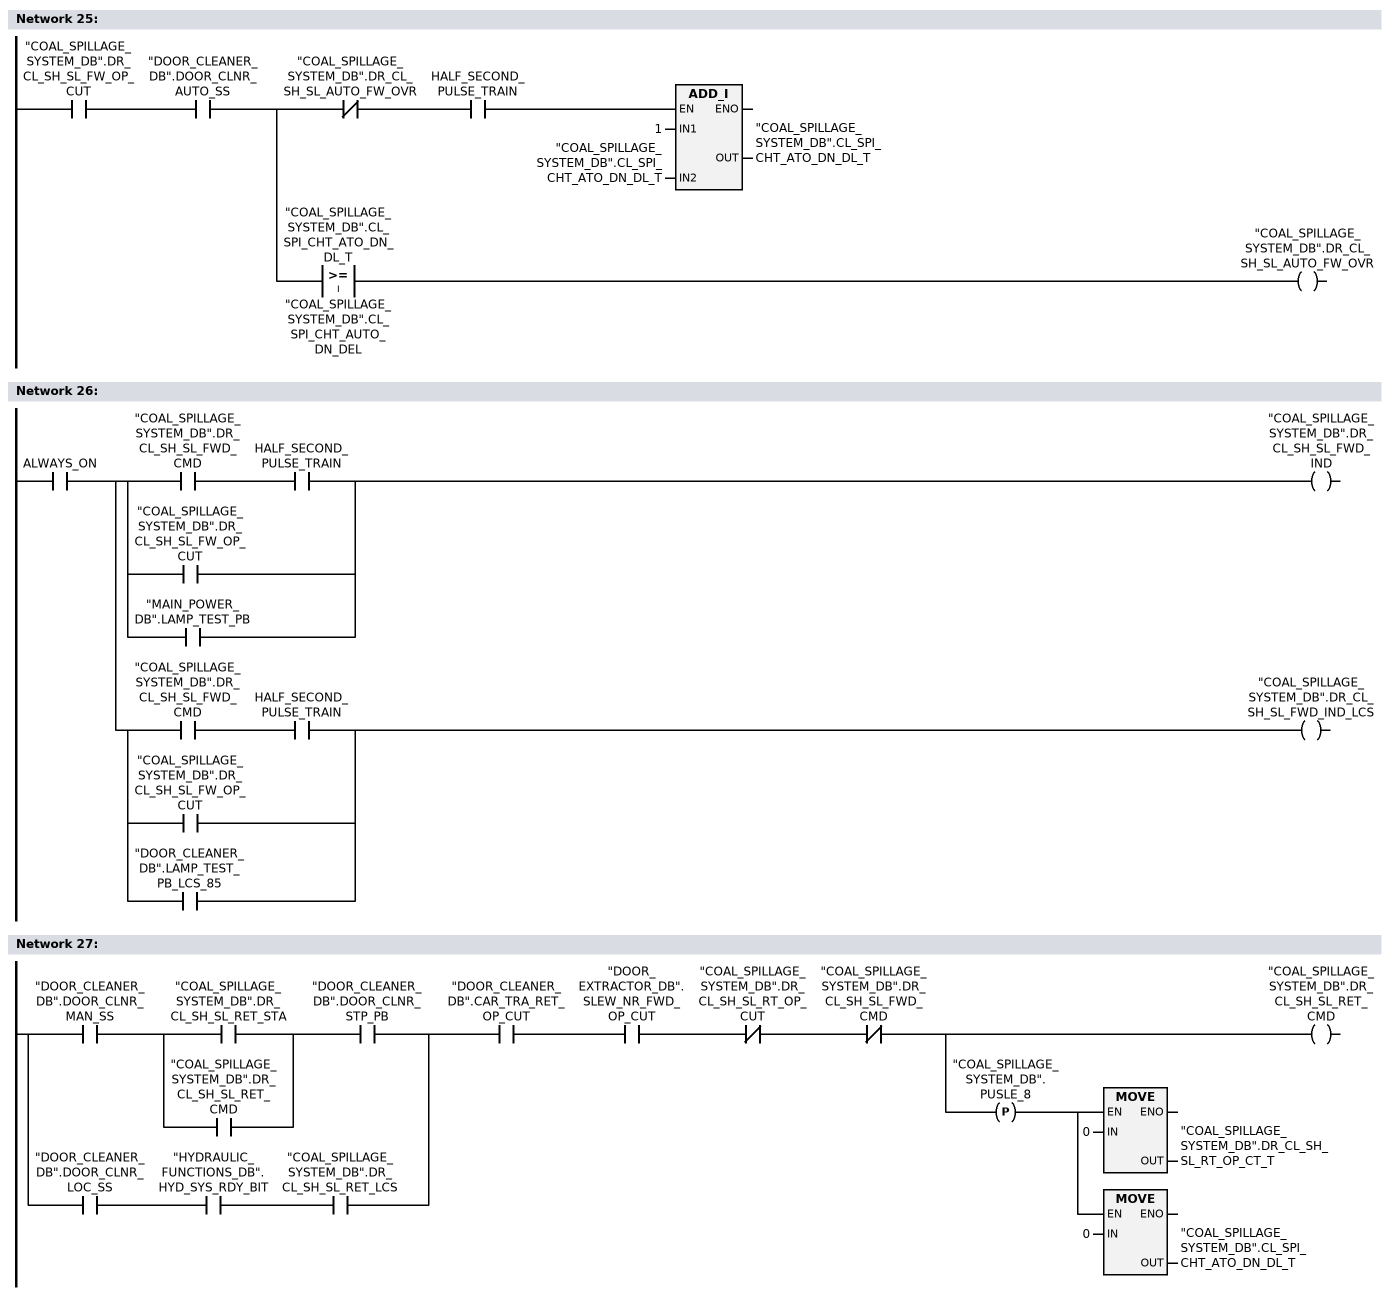
NETWORK
TITLE =
      A     "COAL_SPILLAGE_SYSTEM_DB".DR_CL_SH_SL_FW_OP_CUT;
      A     "DOOR_CLEANER_DB".DOOR_CLNR_AUTO_SS;
      =     L 0.0;
      A     L 0.0;
      AN    "COAL_SPILLAGE_SYSTEM_DB".DR_CL_SH_SL_AUTO_FW_OVR;
      A     "HALF_SECOND_PULSE_TRAIN";
      JNB   M024;
      L     1;
      L     "COAL_SPILLAGE_SYSTEM_DB".CL_SPI_CHT_ATO_DN_DL_T;
      +I;
      T     "COAL_SPILLAGE_SYSTEM_DB".CL_SPI_CHT_ATO_DN_DL_T;
M024: NOP   0;
      A     L 0.0;
      A(;
      L     "COAL_SPILLAGE_SYSTEM_DB".CL_SPI_CHT_ATO_DN_DL_T;
      L     "COAL_SPILLAGE_SYSTEM_DB".CL_SPI_CHT_AUTO_DN_DEL;
      >=I;
      );
      =     "COAL_SPILLAGE_SYSTEM_DB".DR_CL_SH_SL_AUTO_FW_OVR;
NETWORK
TITLE =
      A     "ALWAYS_ON";
      =     L 0.0;
      A     L 0.0;
      A(;
      A     "COAL_SPILLAGE_SYSTEM_DB".DR_CL_SH_SL_FWD_CMD;
      A     "HALF_SECOND_PULSE_TRAIN";
      O     "COAL_SPILLAGE_SYSTEM_DB".DR_CL_SH_SL_FW_OP_CUT;
      O     "MAIN_POWER_DB".LAMP_TEST_PB;
      );
      =     "COAL_SPILLAGE_SYSTEM_DB".DR_CL_SH_SL_FWD_IND;
      A     L 0.0;
      A(;
      A     "COAL_SPILLAGE_SYSTEM_DB".DR_CL_SH_SL_FWD_CMD;
      A     "HALF_SECOND_PULSE_TRAIN";
      O     "COAL_SPILLAGE_SYSTEM_DB".DR_CL_SH_SL_FW_OP_CUT;
      O     "DOOR_CLEANER_DB".LAMP_TEST_PB_LCS_85;
      );
      =     "COAL_SPILLAGE_SYSTEM_DB".DR_CL_SH_SL_FWD_IND_LCS;
NETWORK
TITLE =
      A(;
      A     "DOOR_CLEANER_DB".DOOR_CLNR_MAN_SS;
      A(;
      O     "COAL_SPILLAGE_SYSTEM_DB".DR_CL_SH_SL_RET_STA;
      O     "COAL_SPILLAGE_SYSTEM_DB".DR_CL_SH_SL_RET_CMD;
      );
      A     "DOOR_CLEANER_DB".DOOR_CLNR_STP_PB;
      O;
      A     "DOOR_CLEANER_DB".DOOR_CLNR_LOC_SS;
      A     "HYDRAULIC_FUNCTIONS_DB".HYD_SYS_RDY_BIT;
      A     "COAL_SPILLAGE_SYSTEM_DB".DR_CL_SH_SL_RET_LCS;
      );
      A     "DOOR_CLEANER_DB".CAR_TRA_RET_OP_CUT;
      A     "DOOR_EXTRACTOR_DB".SLEW_NR_FWD_OP_CUT;
      AN    "COAL_SPILLAGE_SYSTEM_DB".DR_CL_SH_SL_RT_OP_CUT;
      AN    "COAL_SPILLAGE_SYSTEM_DB".DR_CL_SH_SL_FWD_CMD;
      =     L 0.0;
      A     L 0.0;
      BLD   102;
      =     "COAL_SPILLAGE_SYSTEM_DB".DR_CL_SH_SL_RET_CMD;
      A     L 0.0;
      FP    "COAL_SPILLAGE_SYSTEM_DB".PUSLE_8;
      =     L 0.1;
      A     L 0.1;
      JNB   M025;
      L     0;
      T     "COAL_SPILLAGE_SYSTEM_DB".DR_CL_SH_SL_RT_OP_CT_T;
M025: NOP   0;
      A     L 0.1;
      JNB   M026;
      L     0;
      T     "COAL_SPILLAGE_SYSTEM_DB".CL_SPI_CHT_ATO_DN_DL_T;
M026: NOP   0;
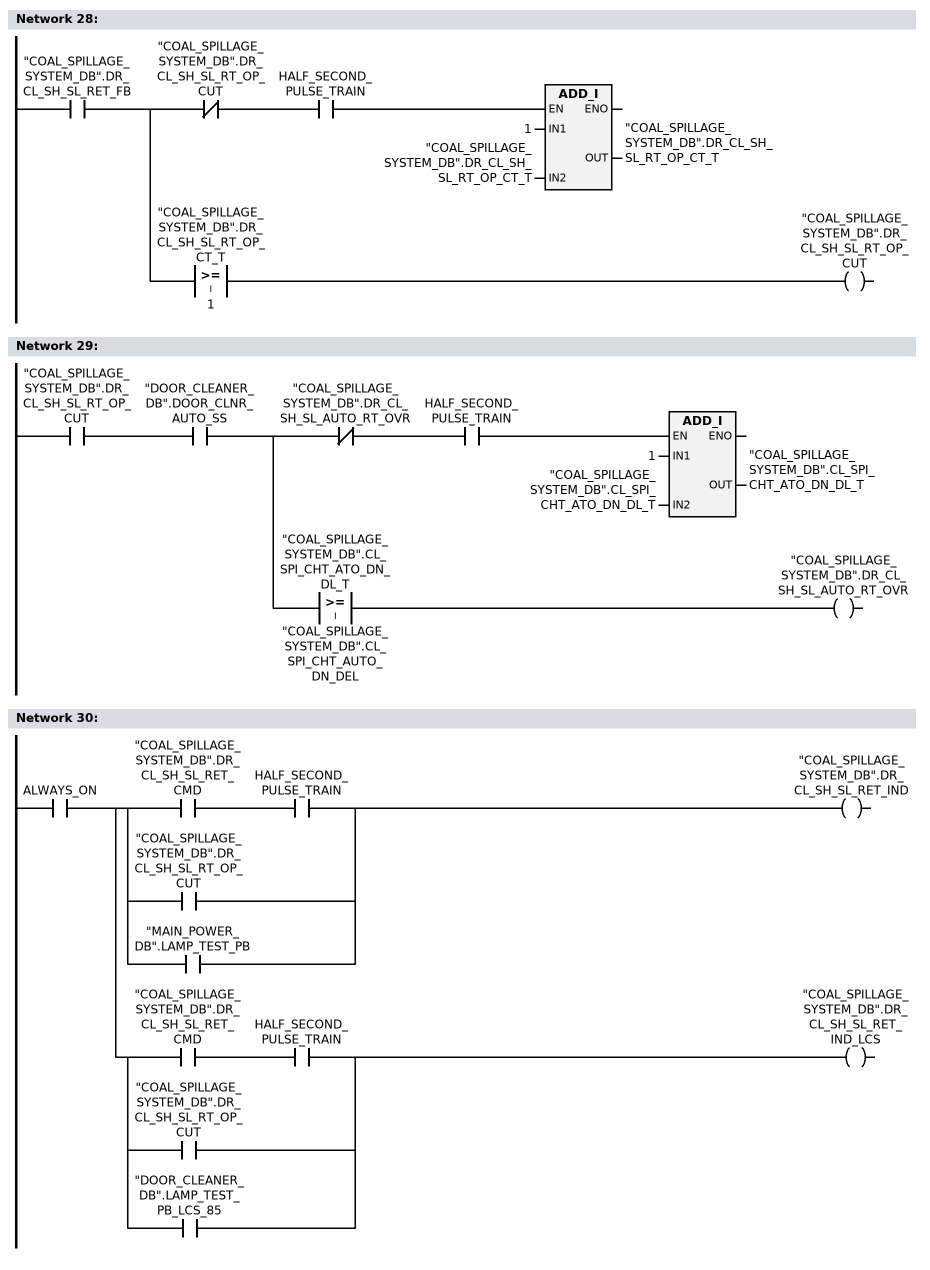
NETWORK
TITLE =
      A     "COAL_SPILLAGE_SYSTEM_DB".DR_CL_SH_SL_RET_FB;
      =     L 0.0;
      A     L 0.0;
      AN    "COAL_SPILLAGE_SYSTEM_DB".DR_CL_SH_SL_RT_OP_CUT;
      A     "HALF_SECOND_PULSE_TRAIN";
      JNB   M027;
      L     1;
      L     "COAL_SPILLAGE_SYSTEM_DB".DR_CL_SH_SL_RT_OP_CT_T;
      +I;
      T     "COAL_SPILLAGE_SYSTEM_DB".DR_CL_SH_SL_RT_OP_CT_T;
M027: NOP   0;
      A     L 0.0;
      A(;
      L     "COAL_SPILLAGE_SYSTEM_DB".DR_CL_SH_SL_RT_OP_CT_T;
      L     1;
      >=I;
      );
      =     "COAL_SPILLAGE_SYSTEM_DB".DR_CL_SH_SL_RT_OP_CUT;
NETWORK
TITLE =
      A     "COAL_SPILLAGE_SYSTEM_DB".DR_CL_SH_SL_RT_OP_CUT;
      A     "DOOR_CLEANER_DB".DOOR_CLNR_AUTO_SS;
      =     L 0.0;
      A     L 0.0;
      AN    "COAL_SPILLAGE_SYSTEM_DB".DR_CL_SH_SL_AUTO_RT_OVR;
      A     "HALF_SECOND_PULSE_TRAIN";
      JNB   M028;
      L     1;
      L     "COAL_SPILLAGE_SYSTEM_DB".CL_SPI_CHT_ATO_DN_DL_T;
      +I;
      T     "COAL_SPILLAGE_SYSTEM_DB".CL_SPI_CHT_ATO_DN_DL_T;
M028: NOP   0;
      A     L 0.0;
      A(;
      L     "COAL_SPILLAGE_SYSTEM_DB".CL_SPI_CHT_ATO_DN_DL_T;
      L     "COAL_SPILLAGE_SYSTEM_DB".CL_SPI_CHT_AUTO_DN_DEL;
      >=I;
      );
      =     "COAL_SPILLAGE_SYSTEM_DB".DR_CL_SH_SL_AUTO_RT_OVR;
NETWORK
TITLE =
      A     "ALWAYS_ON";
      =     L 0.0;
      A     L 0.0;
      A(;
      A     "COAL_SPILLAGE_SYSTEM_DB".DR_CL_SH_SL_RET_CMD;
      A     "HALF_SECOND_PULSE_TRAIN";
      O     "COAL_SPILLAGE_SYSTEM_DB".DR_CL_SH_SL_RT_OP_CUT;
      O     "MAIN_POWER_DB".LAMP_TEST_PB;
      );
      =     "COAL_SPILLAGE_SYSTEM_DB".DR_CL_SH_SL_RET_IND;
      A     L 0.0;
      A(;
      A     "COAL_SPILLAGE_SYSTEM_DB".DR_CL_SH_SL_RET_CMD;
      A     "HALF_SECOND_PULSE_TRAIN";
      O     "COAL_SPILLAGE_SYSTEM_DB".DR_CL_SH_SL_RT_OP_CUT;
      O     "DOOR_CLEANER_DB".LAMP_TEST_PB_LCS_85;
      );
      =     "COAL_SPILLAGE_SYSTEM_DB".DR_CL_SH_SL_RET_IND_LCS;
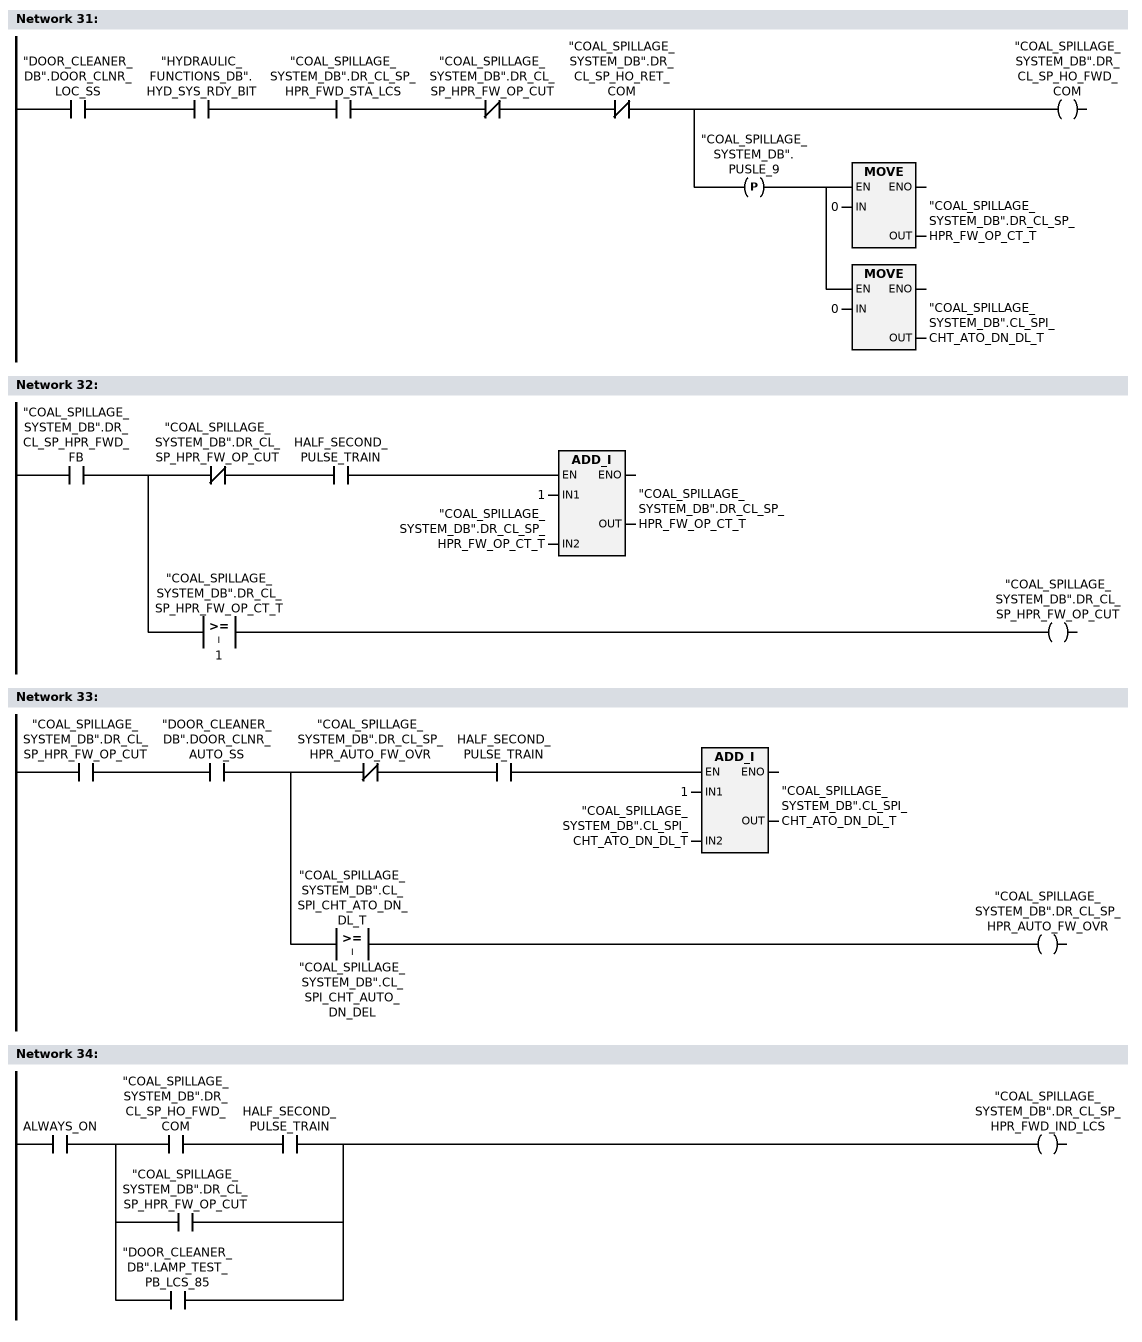
NETWORK
TITLE =
      A     "DOOR_CLEANER_DB".DOOR_CLNR_LOC_SS;
      A     "HYDRAULIC_FUNCTIONS_DB".HYD_SYS_RDY_BIT;
      A     "COAL_SPILLAGE_SYSTEM_DB".DR_CL_SP_HPR_FWD_STA_LCS;
      AN    "COAL_SPILLAGE_SYSTEM_DB".DR_CL_SP_HPR_FW_OP_CUT;
      AN    "COAL_SPILLAGE_SYSTEM_DB".DR_CL_SP_HO_RET_COM;
      =     L 0.0;
      A     L 0.0;
      BLD   102;
      =     "COAL_SPILLAGE_SYSTEM_DB".DR_CL_SP_HO_FWD_COM;
      A     L 0.0;
      FP    "COAL_SPILLAGE_SYSTEM_DB".PUSLE_9;
      =     L 0.1;
      A     L 0.1;
      JNB   M029;
      L     0;
      T     "COAL_SPILLAGE_SYSTEM_DB".DR_CL_SP_HPR_FW_OP_CT_T;
M029: NOP   0;
      A     L 0.1;
      JNB   M030;
      L     0;
      T     "COAL_SPILLAGE_SYSTEM_DB".CL_SPI_CHT_ATO_DN_DL_T;
M030: NOP   0;
NETWORK
TITLE =
      A     "COAL_SPILLAGE_SYSTEM_DB".DR_CL_SP_HPR_FWD_FB;
      =     L 0.0;
      A     L 0.0;
      AN    "COAL_SPILLAGE_SYSTEM_DB".DR_CL_SP_HPR_FW_OP_CUT;
      A     "HALF_SECOND_PULSE_TRAIN";
      JNB   M031;
      L     1;
      L     "COAL_SPILLAGE_SYSTEM_DB".DR_CL_SP_HPR_FW_OP_CT_T;
      +I;
      T     "COAL_SPILLAGE_SYSTEM_DB".DR_CL_SP_HPR_FW_OP_CT_T;
M031: NOP   0;
      A     L 0.0;
      A(;
      L     "COAL_SPILLAGE_SYSTEM_DB".DR_CL_SP_HPR_FW_OP_CT_T;
      L     1;
      >=I;
      );
      =     "COAL_SPILLAGE_SYSTEM_DB".DR_CL_SP_HPR_FW_OP_CUT;
NETWORK
TITLE =
      A     "COAL_SPILLAGE_SYSTEM_DB".DR_CL_SP_HPR_FW_OP_CUT;
      A     "DOOR_CLEANER_DB".DOOR_CLNR_AUTO_SS;
      =     L 0.0;
      A     L 0.0;
      AN    "COAL_SPILLAGE_SYSTEM_DB".DR_CL_SP_HPR_AUTO_FW_OVR;
      A     "HALF_SECOND_PULSE_TRAIN";
      JNB   M032;
      L     1;
      L     "COAL_SPILLAGE_SYSTEM_DB".CL_SPI_CHT_ATO_DN_DL_T;
      +I;
      T     "COAL_SPILLAGE_SYSTEM_DB".CL_SPI_CHT_ATO_DN_DL_T;
M032: NOP   0;
      A     L 0.0;
      A(;
      L     "COAL_SPILLAGE_SYSTEM_DB".CL_SPI_CHT_ATO_DN_DL_T;
      L     "COAL_SPILLAGE_SYSTEM_DB".CL_SPI_CHT_AUTO_DN_DEL;
      >=I;
      );
      =     "COAL_SPILLAGE_SYSTEM_DB".DR_CL_SP_HPR_AUTO_FW_OVR;
NETWORK
TITLE =
      A     "ALWAYS_ON";
      A(;
      A     "COAL_SPILLAGE_SYSTEM_DB".DR_CL_SP_HO_FWD_COM;
      A     "HALF_SECOND_PULSE_TRAIN";
      O     "COAL_SPILLAGE_SYSTEM_DB".DR_CL_SP_HPR_FW_OP_CUT;
      O     "DOOR_CLEANER_DB".LAMP_TEST_PB_LCS_85;
      );
      =     "COAL_SPILLAGE_SYSTEM_DB".DR_CL_SP_HPR_FWD_IND_LCS;
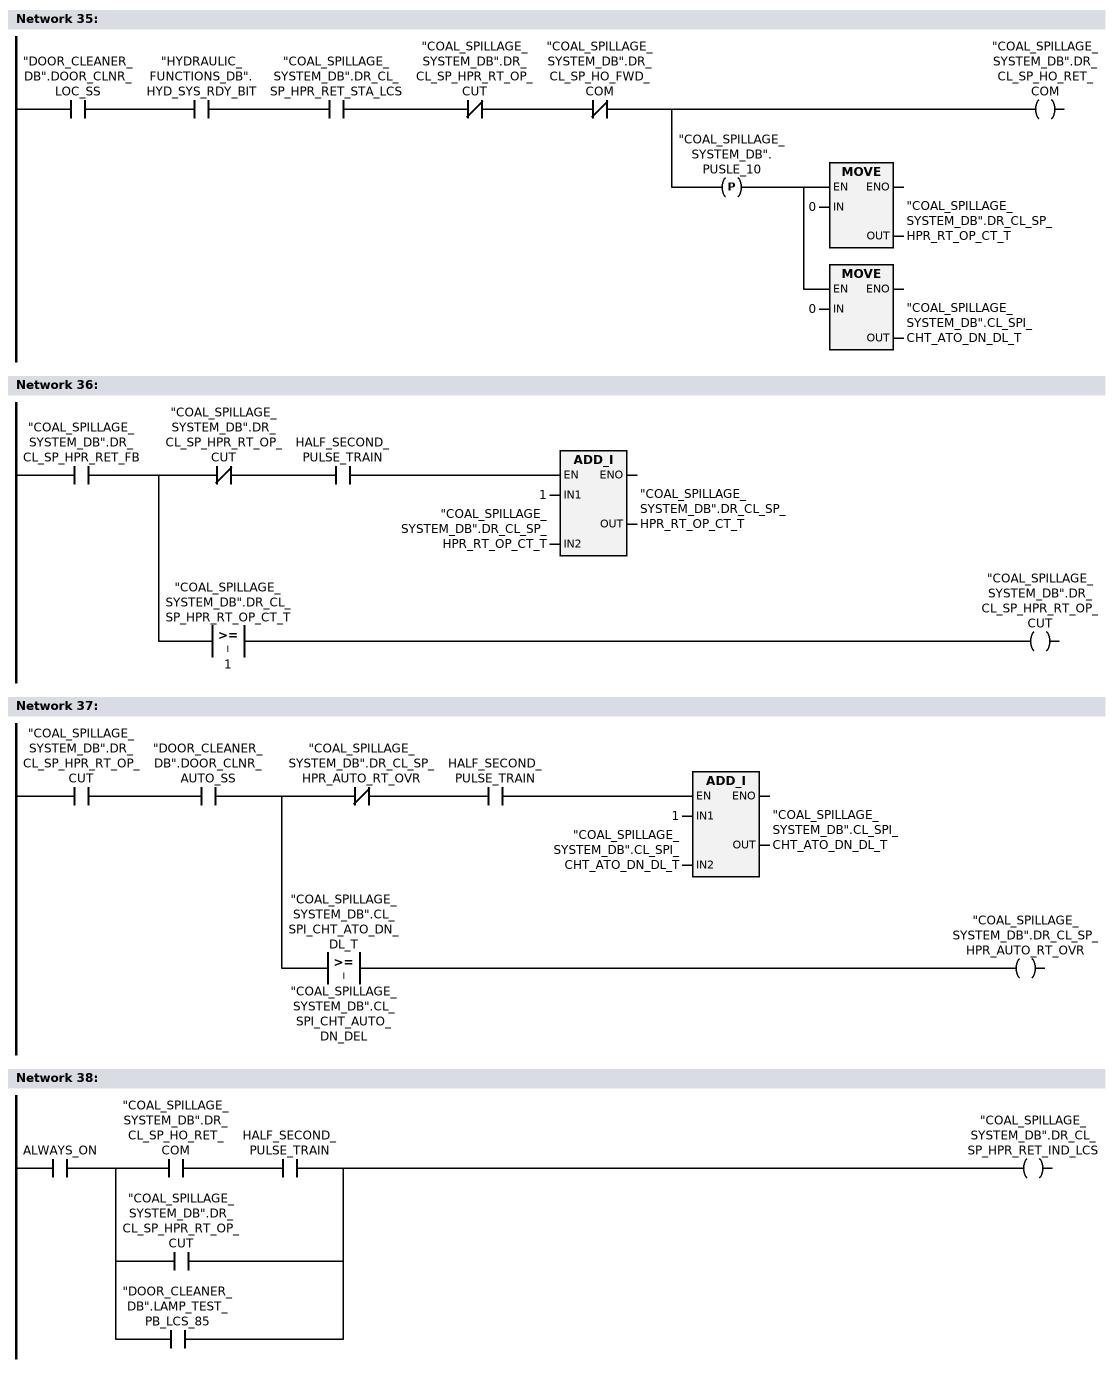
NETWORK
TITLE =
      A     "DOOR_CLEANER_DB".DOOR_CLNR_LOC_SS;
      A     "HYDRAULIC_FUNCTIONS_DB".HYD_SYS_RDY_BIT;
      A     "COAL_SPILLAGE_SYSTEM_DB".DR_CL_SP_HPR_RET_STA_LCS;
      AN    "COAL_SPILLAGE_SYSTEM_DB".DR_CL_SP_HPR_RT_OP_CUT;
      AN    "COAL_SPILLAGE_SYSTEM_DB".DR_CL_SP_HO_FWD_COM;
      =     L 0.0;
      A     L 0.0;
      BLD   102;
      =     "COAL_SPILLAGE_SYSTEM_DB".DR_CL_SP_HO_RET_COM;
      A     L 0.0;
      FP    "COAL_SPILLAGE_SYSTEM_DB".PUSLE_10;
      =     L 0.1;
      A     L 0.1;
      JNB   M033;
      L     0;
      T     "COAL_SPILLAGE_SYSTEM_DB".DR_CL_SP_HPR_RT_OP_CT_T;
M033: NOP   0;
      A     L 0.1;
      JNB   M034;
      L     0;
      T     "COAL_SPILLAGE_SYSTEM_DB".CL_SPI_CHT_ATO_DN_DL_T;
M034: NOP   0;
NETWORK
TITLE =
      A     "COAL_SPILLAGE_SYSTEM_DB".DR_CL_SP_HPR_RET_FB;
      =     L 0.0;
      A     L 0.0;
      AN    "COAL_SPILLAGE_SYSTEM_DB".DR_CL_SP_HPR_RT_OP_CUT;
      A     "HALF_SECOND_PULSE_TRAIN";
      JNB   M035;
      L     1;
      L     "COAL_SPILLAGE_SYSTEM_DB".DR_CL_SP_HPR_RT_OP_CT_T;
      +I;
      T     "COAL_SPILLAGE_SYSTEM_DB".DR_CL_SP_HPR_RT_OP_CT_T;
M035: NOP   0;
      A     L 0.0;
      A(;
      L     "COAL_SPILLAGE_SYSTEM_DB".DR_CL_SP_HPR_RT_OP_CT_T;
      L     1;
      >=I;
      );
      =     "COAL_SPILLAGE_SYSTEM_DB".DR_CL_SP_HPR_RT_OP_CUT;
NETWORK
TITLE =
      A     "COAL_SPILLAGE_SYSTEM_DB".DR_CL_SP_HPR_RT_OP_CUT;
      A     "DOOR_CLEANER_DB".DOOR_CLNR_AUTO_SS;
      =     L 0.0;
      A     L 0.0;
      AN    "COAL_SPILLAGE_SYSTEM_DB".DR_CL_SP_HPR_AUTO_RT_OVR;
      A     "HALF_SECOND_PULSE_TRAIN";
      JNB   M036;
      L     1;
      L     "COAL_SPILLAGE_SYSTEM_DB".CL_SPI_CHT_ATO_DN_DL_T;
      +I;
      T     "COAL_SPILLAGE_SYSTEM_DB".CL_SPI_CHT_ATO_DN_DL_T;
M036: NOP   0;
      A     L 0.0;
      A(;
      L     "COAL_SPILLAGE_SYSTEM_DB".CL_SPI_CHT_ATO_DN_DL_T;
      L     "COAL_SPILLAGE_SYSTEM_DB".CL_SPI_CHT_AUTO_DN_DEL;
      >=I;
      );
      =     "COAL_SPILLAGE_SYSTEM_DB".DR_CL_SP_HPR_AUTO_RT_OVR;
NETWORK
TITLE =
      A     "ALWAYS_ON";
      A(;
      A     "COAL_SPILLAGE_SYSTEM_DB".DR_CL_SP_HO_RET_COM;
      A     "HALF_SECOND_PULSE_TRAIN";
      O     "COAL_SPILLAGE_SYSTEM_DB".DR_CL_SP_HPR_RT_OP_CUT;
      O     "DOOR_CLEANER_DB".LAMP_TEST_PB_LCS_85;
      );
      =     "COAL_SPILLAGE_SYSTEM_DB".DR_CL_SP_HPR_RET_IND_LCS;
END_FUNCTION

FUNCTION "PROFIBUS_COMMUNICATION" : VOID	// FC 19
AUTHOR : Kamillas
VERSION : 0.1
BEGIN
// (block stored without names or comments; labels and parameter names are numbered)
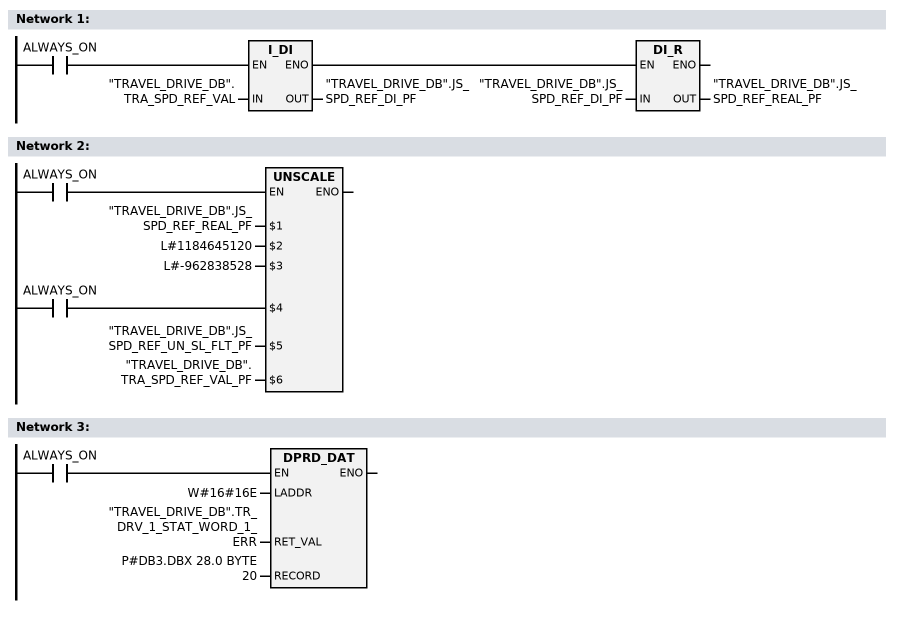
NETWORK
TITLE =
      A(;
      A     "ALWAYS_ON";
      JNB   M001;
      L     "TRAVEL_DRIVE_DB".TRA_SPD_REF_VAL;
      ITD;
      T     "TRAVEL_DRIVE_DB".JS_SPD_REF_DI_PF;
      SET;
      SAVE;
      CLR;
M001: A     BR;
      );
      JNB   M002;
      L     "TRAVEL_DRIVE_DB".JS_SPD_REF_DI_PF;
      DTR;
      T     "TRAVEL_DRIVE_DB".JS_SPD_REF_REAL_PF;
M002: NOP   0;
NETWORK
TITLE =
      A     "ALWAYS_ON";
      =     L 0.0;
      BLD   103;
      A     "ALWAYS_ON";
      JNB   M003;
      CALL  "UNSCALE" (
           $1                       := "TRAVEL_DRIVE_DB".JS_SPD_REF_REAL_PF,
           $2                       := L#1184645120,
           $3                       := L#-962838528,
           $4                       := L 0.0,
           $5                       := "TRAVEL_DRIVE_DB".JS_SPD_REF_UN_SL_FLT_PF,
           $6                       := "TRAVEL_DRIVE_DB".TRA_SPD_REF_VAL_PF);
M003: NOP   0;
NETWORK
TITLE =
      A     "ALWAYS_ON";
      JNB   M004;
      CALL  "DPRD_DAT" (
           LADDR                    := W#16#16E,
           RET_VAL                  := "TRAVEL_DRIVE_DB".TR_DRV_1_STAT_WORD_1_ERR,
           RECORD                   := P#DB3.DBX 28.0 BYTE 20);
M004: NOP   0;
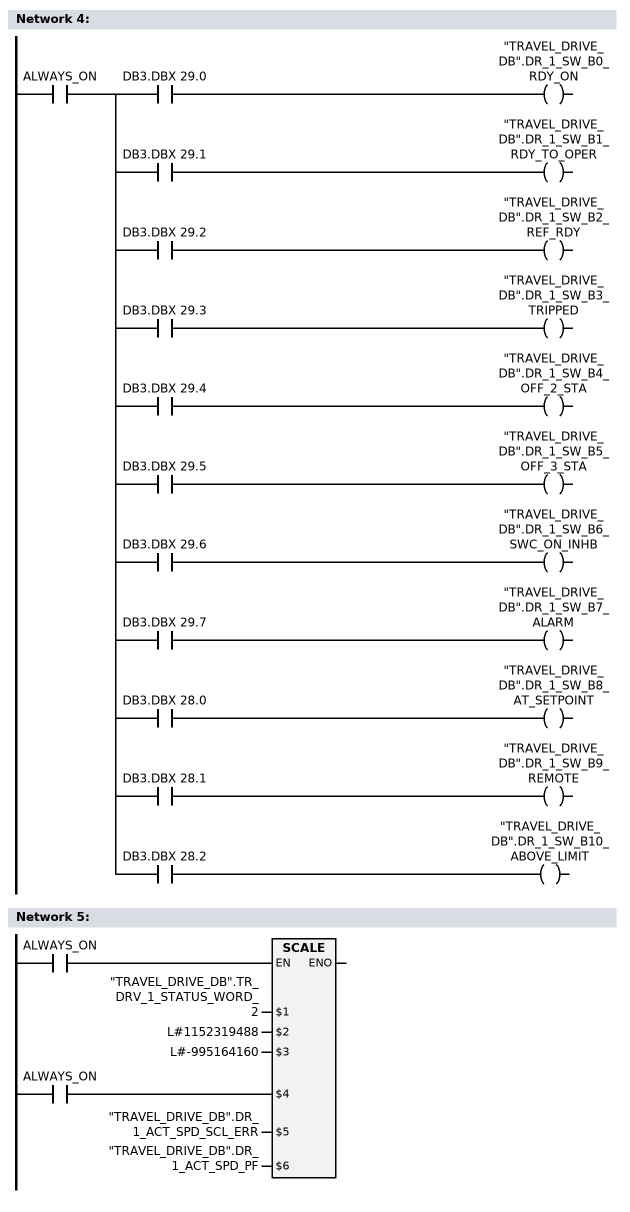
NETWORK
TITLE =
      A     "ALWAYS_ON";
      =     L 0.0;
      A     L 0.0;
      A     DB3.DBX 29.0;
      =     "TRAVEL_DRIVE_DB".DR_1_SW_B0_RDY_ON;
      A     L 0.0;
      A     DB3.DBX 29.1;
      =     "TRAVEL_DRIVE_DB".DR_1_SW_B1_RDY_TO_OPER;
      A     L 0.0;
      A     DB3.DBX 29.2;
      =     "TRAVEL_DRIVE_DB".DR_1_SW_B2_REF_RDY;
      A     L 0.0;
      A     DB3.DBX 29.3;
      =     "TRAVEL_DRIVE_DB".DR_1_SW_B3_TRIPPED;
      A     L 0.0;
      A     DB3.DBX 29.4;
      =     "TRAVEL_DRIVE_DB".DR_1_SW_B4_OFF_2_STA;
      A     L 0.0;
      A     DB3.DBX 29.5;
      =     "TRAVEL_DRIVE_DB".DR_1_SW_B5_OFF_3_STA;
      A     L 0.0;
      A     DB3.DBX 29.6;
      =     "TRAVEL_DRIVE_DB".DR_1_SW_B6_SWC_ON_INHB;
      A     L 0.0;
      A     DB3.DBX 29.7;
      =     "TRAVEL_DRIVE_DB".DR_1_SW_B7_ALARM;
      A     L 0.0;
      A     DB3.DBX 28.0;
      =     "TRAVEL_DRIVE_DB".DR_1_SW_B8_AT_SETPOINT;
      A     L 0.0;
      A     DB3.DBX 28.1;
      =     "TRAVEL_DRIVE_DB".DR_1_SW_B9_REMOTE;
      A     L 0.0;
      A     DB3.DBX 28.2;
      =     "TRAVEL_DRIVE_DB".DR_1_SW_B10_ABOVE_LIMIT;
NETWORK
TITLE =
      A     "ALWAYS_ON";
      =     L 0.0;
      BLD   103;
      A     "ALWAYS_ON";
      JNB   M005;
      CALL  "SCALE" (
           $1                       := "TRAVEL_DRIVE_DB".TR_DRV_1_STATUS_WORD_2,
           $2                       := L#1152319488,
           $3                       := L#-995164160,
           $4                       := L 0.0,
           $5                       := "TRAVEL_DRIVE_DB".DR_1_ACT_SPD_SCL_ERR,
           $6                       := "TRAVEL_DRIVE_DB".DR_1_ACT_SPD_PF);
M005: NOP   0;
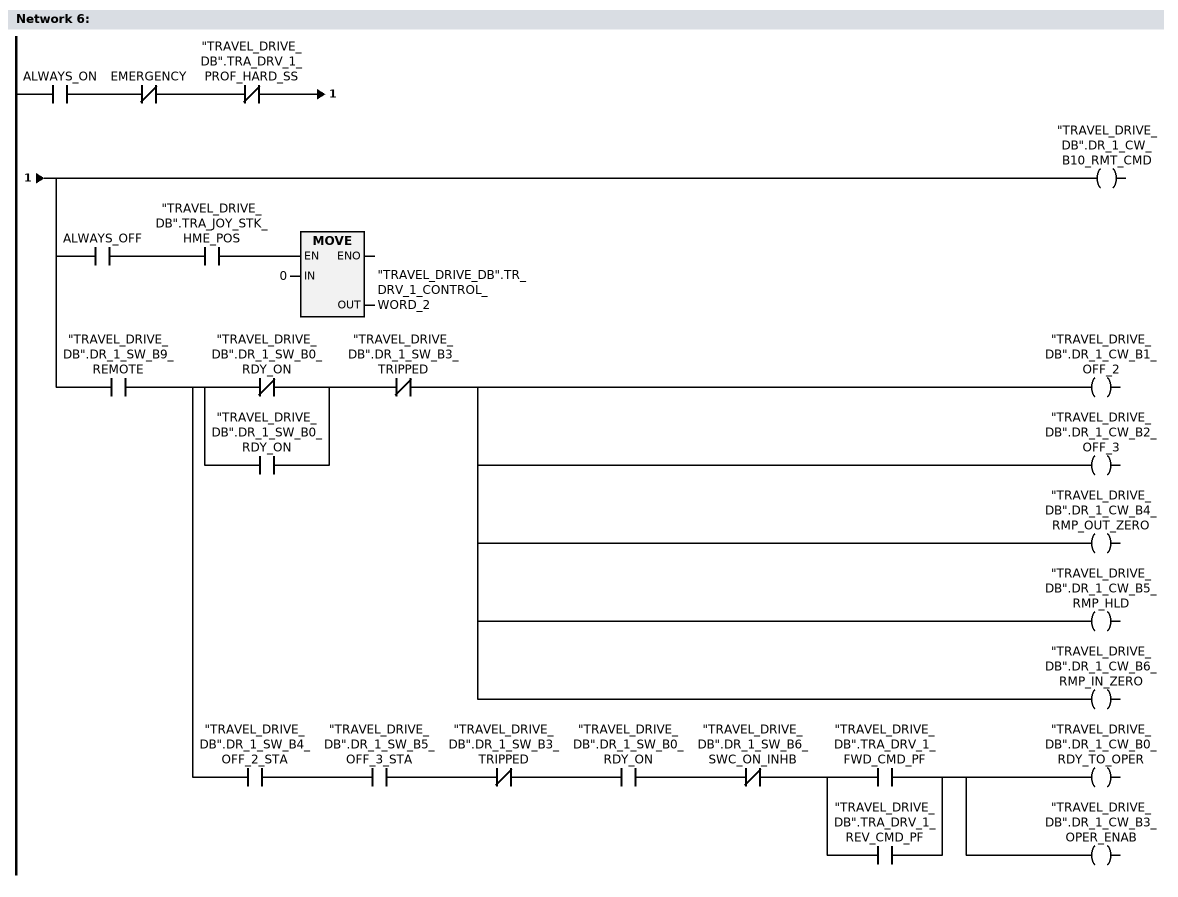
NETWORK
TITLE =
      A     "ALWAYS_ON";
      AN    "EMERGENCY";
      AN    "TRAVEL_DRIVE_DB".TRA_DRV_1_PROF_HARD_SS;
      =     L 0.0;
      A     L 0.0;
      BLD   102;
      =     "TRAVEL_DRIVE_DB".DR_1_CW_B10_RMT_CMD;
      A     L 0.0;
      A     "ALWAYS_OFF";
      A     "TRAVEL_DRIVE_DB".TRA_JOY_STK_HME_POS;
      JNB   M006;
      L     0;
      T     "TRAVEL_DRIVE_DB".TR_DRV_1_CONTROL_WORD_2;
M006: NOP   0;
      A     L 0.0;
      A     "TRAVEL_DRIVE_DB".DR_1_SW_B9_REMOTE;
      =     L 0.1;
      A     L 0.1;
      A(;
      ON    "TRAVEL_DRIVE_DB".DR_1_SW_B0_RDY_ON;
      O     "TRAVEL_DRIVE_DB".DR_1_SW_B0_RDY_ON;
      );
      AN    "TRAVEL_DRIVE_DB".DR_1_SW_B3_TRIPPED;
      =     "TRAVEL_DRIVE_DB".DR_1_CW_B1_OFF_2;
      =     "TRAVEL_DRIVE_DB".DR_1_CW_B2_OFF_3;
      =     "TRAVEL_DRIVE_DB".DR_1_CW_B4_RMP_OUT_ZERO;
      =     "TRAVEL_DRIVE_DB".DR_1_CW_B5_RMP_HLD;
      =     "TRAVEL_DRIVE_DB".DR_1_CW_B6_RMP_IN_ZERO;
      A     L 0.1;
      A     "TRAVEL_DRIVE_DB".DR_1_SW_B4_OFF_2_STA;
      A     "TRAVEL_DRIVE_DB".DR_1_SW_B5_OFF_3_STA;
      AN    "TRAVEL_DRIVE_DB".DR_1_SW_B3_TRIPPED;
      A     "TRAVEL_DRIVE_DB".DR_1_SW_B0_RDY_ON;
      AN    "TRAVEL_DRIVE_DB".DR_1_SW_B6_SWC_ON_INHB;
      A(;
      O     "TRAVEL_DRIVE_DB".TRA_DRV_1_FWD_CMD_PF;
      O     "TRAVEL_DRIVE_DB".TRA_DRV_1_REV_CMD_PF;
      );
      =     "TRAVEL_DRIVE_DB".DR_1_CW_B0_RDY_TO_OPER;
      =     "TRAVEL_DRIVE_DB".DR_1_CW_B3_OPER_ENAB;
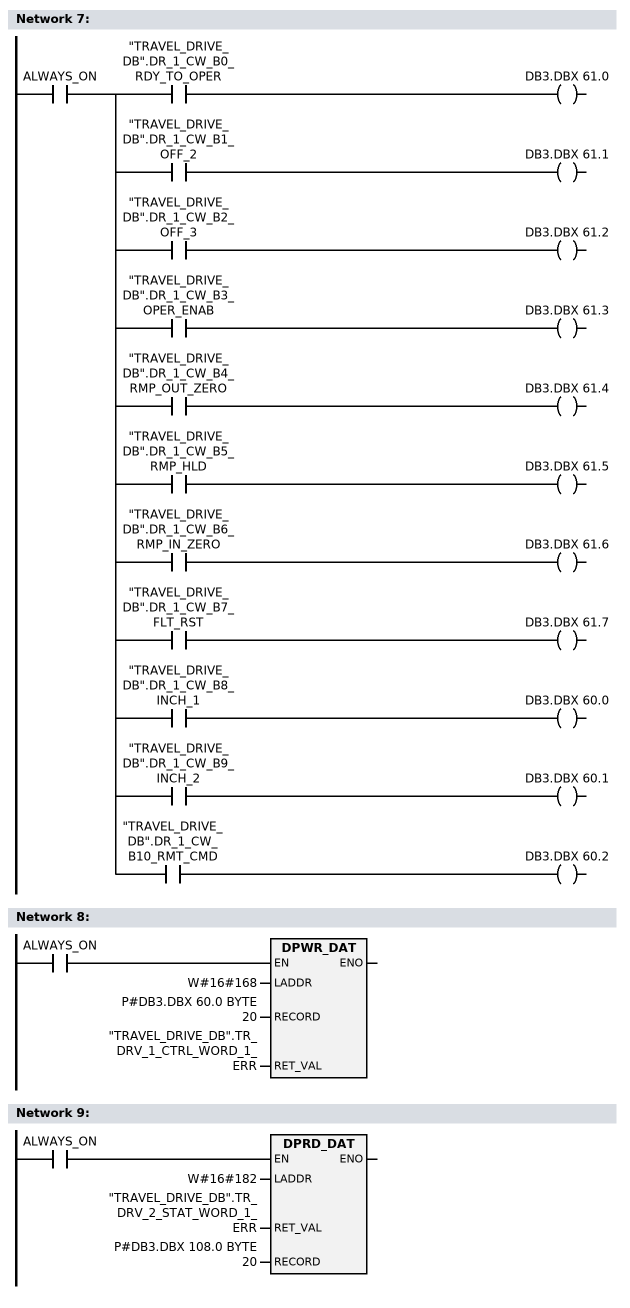
NETWORK
TITLE =
      A     "ALWAYS_ON";
      =     L 0.0;
      A     L 0.0;
      A     "TRAVEL_DRIVE_DB".DR_1_CW_B0_RDY_TO_OPER;
      =     DB3.DBX 61.0;
      A     L 0.0;
      A     "TRAVEL_DRIVE_DB".DR_1_CW_B1_OFF_2;
      =     DB3.DBX 61.1;
      A     L 0.0;
      A     "TRAVEL_DRIVE_DB".DR_1_CW_B2_OFF_3;
      =     DB3.DBX 61.2;
      A     L 0.0;
      A     "TRAVEL_DRIVE_DB".DR_1_CW_B3_OPER_ENAB;
      =     DB3.DBX 61.3;
      A     L 0.0;
      A     "TRAVEL_DRIVE_DB".DR_1_CW_B4_RMP_OUT_ZERO;
      =     DB3.DBX 61.4;
      A     L 0.0;
      A     "TRAVEL_DRIVE_DB".DR_1_CW_B5_RMP_HLD;
      =     DB3.DBX 61.5;
      A     L 0.0;
      A     "TRAVEL_DRIVE_DB".DR_1_CW_B6_RMP_IN_ZERO;
      =     DB3.DBX 61.6;
      A     L 0.0;
      A     "TRAVEL_DRIVE_DB".DR_1_CW_B7_FLT_RST;
      =     DB3.DBX 61.7;
      A     L 0.0;
      A     "TRAVEL_DRIVE_DB".DR_1_CW_B8_INCH_1;
      =     DB3.DBX 60.0;
      A     L 0.0;
      A     "TRAVEL_DRIVE_DB".DR_1_CW_B9_INCH_2;
      =     DB3.DBX 60.1;
      A     L 0.0;
      A     "TRAVEL_DRIVE_DB".DR_1_CW_B10_RMT_CMD;
      =     DB3.DBX 60.2;
NETWORK
TITLE =
      A     "ALWAYS_ON";
      JNB   M007;
      CALL  "DPWR_DAT" (
           LADDR                    := W#16#168,
           RECORD                   := P#DB3.DBX 60.0 BYTE 20,
           RET_VAL                  := "TRAVEL_DRIVE_DB".TR_DRV_1_CTRL_WORD_1_ERR);
M007: NOP   0;
NETWORK
TITLE =
      A     "ALWAYS_ON";
      JNB   M008;
      CALL  "DPRD_DAT" (
           LADDR                    := W#16#182,
           RET_VAL                  := "TRAVEL_DRIVE_DB".TR_DRV_2_STAT_WORD_1_ERR,
           RECORD                   := P#DB3.DBX 108.0 BYTE 20);
M008: NOP   0;
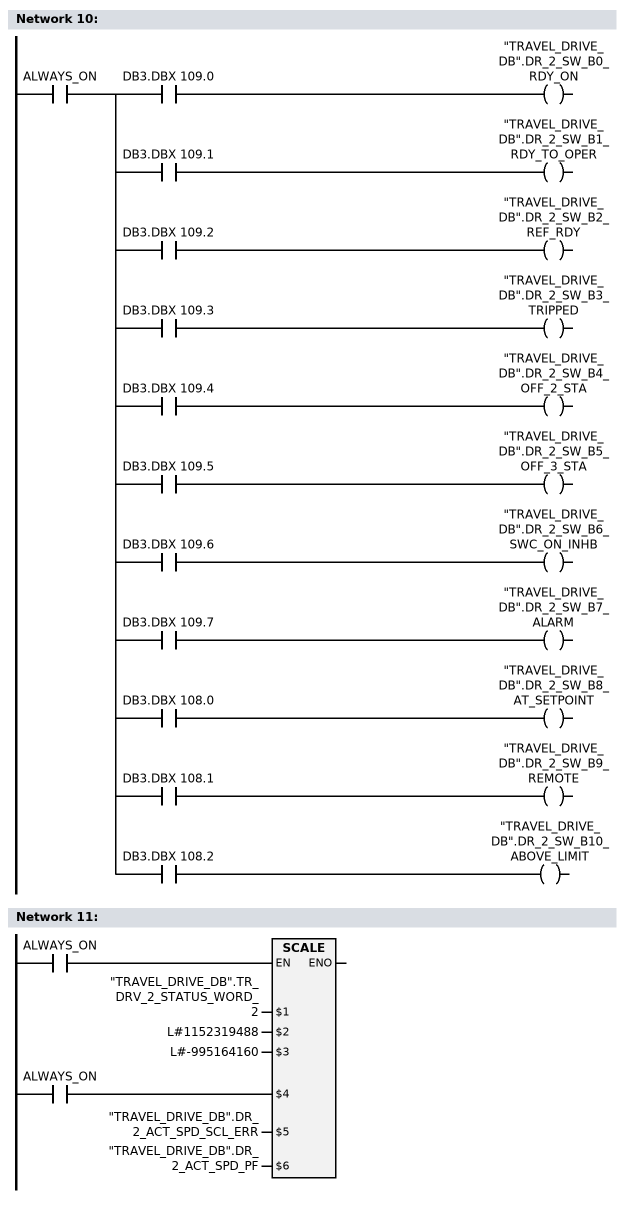
NETWORK
TITLE =
      A     "ALWAYS_ON";
      =     L 0.0;
      A     L 0.0;
      A     DB3.DBX 109.0;
      =     "TRAVEL_DRIVE_DB".DR_2_SW_B0_RDY_ON;
      A     L 0.0;
      A     DB3.DBX 109.1;
      =     "TRAVEL_DRIVE_DB".DR_2_SW_B1_RDY_TO_OPER;
      A     L 0.0;
      A     DB3.DBX 109.2;
      =     "TRAVEL_DRIVE_DB".DR_2_SW_B2_REF_RDY;
      A     L 0.0;
      A     DB3.DBX 109.3;
      =     "TRAVEL_DRIVE_DB".DR_2_SW_B3_TRIPPED;
      A     L 0.0;
      A     DB3.DBX 109.4;
      =     "TRAVEL_DRIVE_DB".DR_2_SW_B4_OFF_2_STA;
      A     L 0.0;
      A     DB3.DBX 109.5;
      =     "TRAVEL_DRIVE_DB".DR_2_SW_B5_OFF_3_STA;
      A     L 0.0;
      A     DB3.DBX 109.6;
      =     "TRAVEL_DRIVE_DB".DR_2_SW_B6_SWC_ON_INHB;
      A     L 0.0;
      A     DB3.DBX 109.7;
      =     "TRAVEL_DRIVE_DB".DR_2_SW_B7_ALARM;
      A     L 0.0;
      A     DB3.DBX 108.0;
      =     "TRAVEL_DRIVE_DB".DR_2_SW_B8_AT_SETPOINT;
      A     L 0.0;
      A     DB3.DBX 108.1;
      =     "TRAVEL_DRIVE_DB".DR_2_SW_B9_REMOTE;
      A     L 0.0;
      A     DB3.DBX 108.2;
      =     "TRAVEL_DRIVE_DB".DR_2_SW_B10_ABOVE_LIMIT;
NETWORK
TITLE =
      A     "ALWAYS_ON";
      =     L 0.0;
      BLD   103;
      A     "ALWAYS_ON";
      JNB   M009;
      CALL  "SCALE" (
           $1                       := "TRAVEL_DRIVE_DB".TR_DRV_2_STATUS_WORD_2,
           $2                       := L#1152319488,
           $3                       := L#-995164160,
           $4                       := L 0.0,
           $5                       := "TRAVEL_DRIVE_DB".DR_2_ACT_SPD_SCL_ERR,
           $6                       := "TRAVEL_DRIVE_DB".DR_2_ACT_SPD_PF);
M009: NOP   0;
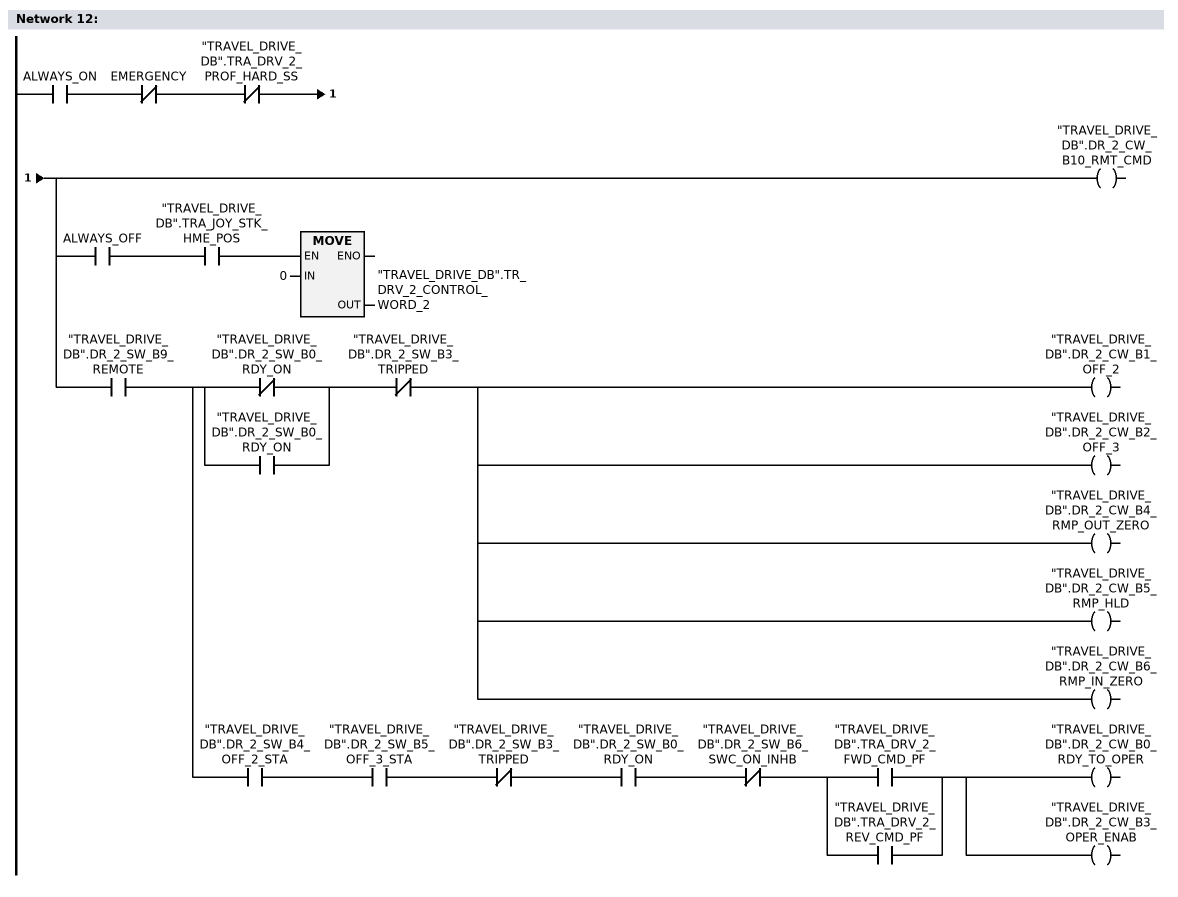
NETWORK
TITLE =
      A     "ALWAYS_ON";
      AN    "EMERGENCY";
      AN    "TRAVEL_DRIVE_DB".TRA_DRV_2_PROF_HARD_SS;
      =     L 0.0;
      A     L 0.0;
      BLD   102;
      =     "TRAVEL_DRIVE_DB".DR_2_CW_B10_RMT_CMD;
      A     L 0.0;
      A     "ALWAYS_OFF";
      A     "TRAVEL_DRIVE_DB".TRA_JOY_STK_HME_POS;
      JNB   M010;
      L     0;
      T     "TRAVEL_DRIVE_DB".TR_DRV_2_CONTROL_WORD_2;
M010: NOP   0;
      A     L 0.0;
      A     "TRAVEL_DRIVE_DB".DR_2_SW_B9_REMOTE;
      =     L 0.1;
      A     L 0.1;
      A(;
      ON    "TRAVEL_DRIVE_DB".DR_2_SW_B0_RDY_ON;
      O     "TRAVEL_DRIVE_DB".DR_2_SW_B0_RDY_ON;
      );
      AN    "TRAVEL_DRIVE_DB".DR_2_SW_B3_TRIPPED;
      =     "TRAVEL_DRIVE_DB".DR_2_CW_B1_OFF_2;
      =     "TRAVEL_DRIVE_DB".DR_2_CW_B2_OFF_3;
      =     "TRAVEL_DRIVE_DB".DR_2_CW_B4_RMP_OUT_ZERO;
      =     "TRAVEL_DRIVE_DB".DR_2_CW_B5_RMP_HLD;
      =     "TRAVEL_DRIVE_DB".DR_2_CW_B6_RMP_IN_ZERO;
      A     L 0.1;
      A     "TRAVEL_DRIVE_DB".DR_2_SW_B4_OFF_2_STA;
      A     "TRAVEL_DRIVE_DB".DR_2_SW_B5_OFF_3_STA;
      AN    "TRAVEL_DRIVE_DB".DR_2_SW_B3_TRIPPED;
      A     "TRAVEL_DRIVE_DB".DR_2_SW_B0_RDY_ON;
      AN    "TRAVEL_DRIVE_DB".DR_2_SW_B6_SWC_ON_INHB;
      A(;
      O     "TRAVEL_DRIVE_DB".TRA_DRV_2_FWD_CMD_PF;
      O     "TRAVEL_DRIVE_DB".TRA_DRV_2_REV_CMD_PF;
      );
      =     "TRAVEL_DRIVE_DB".DR_2_CW_B0_RDY_TO_OPER;
      =     "TRAVEL_DRIVE_DB".DR_2_CW_B3_OPER_ENAB;
